	      //Get Index List was successful
	      IF #instOpcUaNamespaceGIL.Done THEN
	        //Check StatusList
	        FOR #tempIndex := 0 TO UDINT_TO_INT(CountOfElements(#namespaceUris) - 1) DO
	          IF #statOpcUaStatusLists.#namespaceGIL[#tempIndex] <> 16#0 THEN
	            #statOpcUaRequests.NGIL := FALSE;
	            // => OUT
	            #statDiagnostics.status := #ERR_NGIL_SL;
	            #statDiagnostics.subfunctionStatus := #statOpcUaStatusLists.namespaceGIL[#tempIndex];
	            // error during NGIL call --> connection establishment failed
	            #statState := #STATE_CONNECT;
	            EXIT;
	          END_IF;
	        END_FOR;
	        #statOpcUaRequests.NGIL := FALSE;
	        IF NOT #statDiagnostics.status.%X15 THEN
	          //Count up statNamespaceGetIndexCount
	          #statDiagCounter.NamespaceReg += 1;
	          //statNamespaceIndexesSet
	          #statRegisteredLists.NamespaceIndexes := TRUE;
	          //=>OUT
	          //Next Step
	          #statState := #STATE_NODE_GET_HANDLE_LIST;
	        ELSE
	          #statCheckConnectionStatus := TRUE;
	        END_IF;
	      END_IF;
	    END_REGION
	    
	  #STATE_NODE_GET_HANDLE_LIST:
	    REGION Handle NodeId lists
	      //Trigger NodeHandleList SFBs
	      IF NOT #statRegisteredLists.Write AND #writeNodeIds <> NULL AND #writeNodeHdls <> NULL THEN
	        #statOpcUaRequests.writeGHL := TRUE;
	        #statDiagnostics.status := #STATUS_BUSY;
	      ELSE
	        IF NOT #statRegisteredLists.Read AND #readNodeIds <> NULL AND #readNodeHdls <> NULL THEN
	          #statOpcUaRequests.readGHL := TRUE;
	          #statDiagnostics.status := #STATUS_BUSY;
	        ELSE
	          IF NOT #statRegisteredLists.Methods AND #methodNodeIds <> NULL AND #methodHdls <> NULL AND #objNodeIds <> NULL THEN
	            #statOpcUaRequests.methodsGHL := TRUE;
	            #statDiagnostics.status := #STATUS_BUSY;
	          ELSE
	            #statState := #STATE_CONNECTED;
	            #statBusy := FALSE;
	            #statDiagnostics.status := #STATUS_IDLE;
	          END_IF;
	        END_IF;
	      END_IF;
	      
	      REGION Handle ReadList
	        //Read Node Get Handle List was not successful
	        IF #InstOpcUaGHLRead.Error THEN
	          //--> Call ConnectionGetStatus if Status = "16#800D0000"
	          IF #InstOpcUaGHLRead.Status = #STATUS_SERVER_NOT_CONNECTED THEN
	            #statCheckConnectionStatus := TRUE;
	          ELSE
	            //#statCase := #STATE_CONNECT;
	            #statState := #STATE_CONNECTED;
	          END_IF;
	          #statOpcUaRequests.readGHL := FALSE;
	          // => OUT
	          #statDiagnostics.status := #ERR_R_GHL;
	          #statDiagnostics.subfunctionStatus := #InstOpcUaGHLRead.Status;
	        END_IF;
	        
	        //Read Node Get Handle List was successful
	        IF #InstOpcUaGHLRead.Done THEN
	          //Check StatusList
	          FOR #tempIndex := 0 TO UDINT_TO_INT(CountOfElements(#readNodeIds) - 1) DO
	            IF #statOpcUaStatusLists.#readGHL[#tempIndex] <> 16#0 THEN
	              // => OUT
	              #statBusy := FALSE;
	              #statDiagnostics.status := #ERR_R_GHL_SL;
	              #statDiagnostics.subfunctionStatus := #statOpcUaStatusLists.#readGHL[#tempIndex];
	              EXIT;
	            END_IF;
	          END_FOR;
	          #statOpcUaRequests.readGHL := FALSE;
	          // Count up statRegisterCount
	          #statDiagCounter.RegisterRead += 1;
	          // Nodes are registered
	          #statRegisteredLists.Read := TRUE;
	        END_IF;
	      END_REGION
	      REGION Handle Write List
	        //Write Node Get Handle List was not successful
	        IF #instOpcUaGHLWrite.Error THEN
	          //--> Call ConnectionGetStatus if Status = "16#800D0000"
	          IF #instOpcUaGHLWrite.Status = #STATUS_SERVER_NOT_CONNECTED THEN
	            #statCheckConnectionStatus := TRUE;
	          ELSE
	            //#statCase := #STATE_CONNECT;
	            #statState := #STATE_CONNECTED;
	          END_IF;
	          #statOpcUaRequests.writeGHL := FALSE;
	          // => OUT
	          #statDiagnostics.status := #ERR_W_GHL;
	          #statDiagnostics.subfunctionStatus := #instOpcUaGHLWrite.Status;
	        END_IF;
	        
	        //Write Node Get Handle List was successful
	        IF #instOpcUaGHLWrite.Done THEN
	          //Check StatusList
	          FOR #tempIndex := 0 TO UDINT_TO_INT(CountOfElements(#writeNodeIds) - 1) DO
	            IF #statOpcUaStatusLists.#writeGHL[#tempIndex] <> 16#0 THEN
	              // => OUT
	              #statBusy := FALSE;
	              #statDiagnostics.status := #ERR_W_GHL_SL;
	              #statDiagnostics.subfunctionStatus := #statOpcUaStatusLists.#writeGHL[#tempIndex];
	              //#statCase := #STATE_CONNECT;
	              EXIT;
	            END_IF;
	          END_FOR;
	          #statOpcUaRequests.writeGHL := FALSE;
	          // Count up statRegisterCount
	          #statDiagCounter.RegisterWrite += 1;
	          // Nodes are registered
	          #statRegisteredLists.Write := TRUE;
	        END_IF;
	      END_REGION
	      
	      REGION Handle MethodList
	        //Method Get HandleList was not successful
	        IF #instOpcUaGHLMethods.Error THEN
	          //--> Call ConnectionGetStatus if Status = "16#800D0000"
	          IF #instOpcUaGHLMethods.Status = #STATUS_SERVER_NOT_CONNECTED THEN
	            #statCheckConnectionStatus := TRUE;
	          ELSE
	            //#statCase := #STATE_CONNECT;
	            #statState := #STATE_CONNECTED;
	          END_IF;
	          #statOpcUaRequests.methodsGHL := FALSE;
	          // => OUT
	          #statDiagnostics.status := #ERR_M_GHL;
	          #statDiagnostics.subfunctionStatus := #instOpcUaGHLMethods.Status;
	        END_IF;
	        
	        //Method Get Handle List was successful
	        IF #instOpcUaGHLMethods.Done THEN
	          //Check StatusList
	          FOR #tempIndex := 0 TO UDINT_TO_INT(CountOfElements(#methodNodeIds) - 1) DO
	            IF #statOpcUaStatusLists.#methodGHL[#tempIndex] <> 16#0 THEN
	              // => OUT
	              #statBusy := FALSE;
	              #statDiagnostics.status := #ERR_M_GHL_SL;
	              #statDiagnostics.subfunctionStatus := #statOpcUaStatusLists.#methodGHL[#tempIndex];
	              EXIT;
	            END_IF;
	          END_FOR;
	          #statOpcUaRequests.methodsGHL := FALSE;
	          // Count up statRegisterCount
	          #statDiagCounter.RegisterMethods += 1;
	          // Nodes are registered
	          #statRegisteredLists.Methods := TRUE;
	        END_IF;
	      END_REGION
	      
	    END_REGION
	    
	  #STATE_CONNECTED:
	    
	    REGION Command and Idle
	      //Idle as long as no Command was triggered
	      IF NOT #statBusy AND NOT #read AND NOT #write AND NOT #callMethod AND NOT #statCheckConnectionStatus THEN
	        #statDone := FALSE;
	        #statDiagnostics.status := #STATUS_IDLE;
	      END_IF;
	      //OPC_UA_GetStatus function is called cyclically, so the connection is monitored
	      #instCycDiag.TON(IN := NOT #statCycDiagTrigger,
	                       PT := #CYC_TIME_GCS);
	      #statCycDiagTrigger := FALSE;
	      IF #instCycDiag.Q AND NOT #statRHLTrigger AND NOT #tempDisconnectTrigger THEN
	        #statCheckConnectionStatus := TRUE;
	        #statCycDiagTrigger := TRUE;
	      END_IF;
	      
	      REGION Read
	        //Trigger if nodes are registered
	        IF #statRegisteredLists.Read AND #statConnected THEN
	          #tempReadTrigger := #read AND NOT #statOldTriggers.read;
	          #statOldTriggers.read := #read;
	        ELSE
	          IF #read AND #statConnected THEN
	            #statDiagnostics.status := #ERR_RL_NOTREG; //Error no ReadList is registerd Request denied
	            #statDiagnostics.subfunctionStatus := #STATUS_NOT_REGISTERED;
	          ELSE
	            IF NOT #statCheckConnectionStatus THEN
	              #statDiagnostics.status := #STATUS_IDLE; //Wait for Connection Get Status
	            END_IF;
	          END_IF;
	        END_IF;
	        
	        IF #tempReadTrigger THEN
	          #statOpcUaRequests.read := TRUE;
	          #statBusy := TRUE;
	          #statDiagnostics.status := #STATUS_BUSY;
	        ELSE
	          #statOpcUaRequests.read := FALSE;
	        END_IF;
	        //Error
	        IF #instOpcUaReadList.Error THEN
	          //--> Call ConnectionGetStatus if Status = "16#800D0000"
	          IF #instOpcUaReadList.Status = #STATUS_SERVER_NOT_CONNECTED THEN
	            #statCheckConnectionStatus := TRUE;
	          END_IF;
	          #statOpcUaRequests.read := FALSE;
	          // => OUT
	          #statBusy := FALSE;
	          #statDiagnostics.status := #ERR_RL;
	          #statDiagnostics.subfunctionStatus := #instOpcUaReadList.Status;
	        END_IF;
	        
	        //Done
	        IF #instOpcUaReadList.Done THEN
	          //Check StatusList
	          FOR #tempIndex := 0 TO UDINT_TO_INT(CountOfElements(#readNodeIds) - 1) DO
	            IF #statOpcUaStatusLists.#readList[#tempIndex] <> 16#0 THEN
	              // => OUT
	              #statDone := FALSE;
	              #statBusy := FALSE;
	              #statDiagnostics.status := #ERR_RL_SL;
	              #statDiagnostics.subfunctionStatus := #statOpcUaStatusLists.readList[#tempIndex];
	              EXIT;
	            END_IF;
	          END_FOR;
	          #statOpcUaRequests.read := FALSE;
	          // => OUT
	          IF NOT #statDiagnostics.status.%X15 THEN
	            #statDone := TRUE;
	            #statBusy := FALSE;
	            #statDiagnostics.status := #STATUS_DONE;
	            //Count up statReadCount
	            #statDiagCounter.Read += 1;
	            //--> Nodes are read continously ...
	          END_IF;
	        END_IF;
	      END_REGION
	      
	      REGION Write
	        //Trigger if nodes are registered
	        IF #statRegisteredLists.Write AND #statConnected THEN
	          #tempWriteTrigger := #write AND NOT #statOldTriggers.write;
	          #statOldTriggers.write := #write;
	        ELSE
	          IF #write AND #statConnected THEN
	            #statDiagnostics.status := #ERR_WL_NOTREG; //Error no WriteList is registerd Request denied
	            #statDiagnostics.subfunctionStatus := #STATUS_NOT_REGISTERED;
	          ELSE
	            IF NOT #statCheckConnectionStatus THEN
	              #statDiagnostics.status := #STATUS_IDLE; //Wait for Connection Get Status
	            END_IF;
	          END_IF;
	        END_IF;
	        
	        IF #tempWriteTrigger THEN
	          #statOpcUaRequests.write := TRUE;
	          #statBusy := TRUE;
	          #statDiagnostics.status := #STATUS_BUSY;
	        ELSE
	          #statOpcUaRequests.write := FALSE;
	        END_IF;
	        //Error
	        IF #instOpcUaWriteList.Error THEN
	          //--> Call ConnectionGetStatus if Status = "16#800D0000"
	          IF #instOpcUaWriteList.Status = #STATUS_SERVER_NOT_CONNECTED THEN
	            #statCheckConnectionStatus := TRUE;
	          END_IF;
	          #statOpcUaRequests.write := FALSE;
	          // => OUT
	          #statBusy := FALSE;
	          #statDiagnostics.status := #ERR_WL;
	          #statDiagnostics.subfunctionStatus := #instOpcUaWriteList.Status;
	        END_IF;
	        
	        //Done
	        IF #instOpcUaWriteList.Done THEN
	          //Check StatusList
	          FOR #tempIndex := 0 TO UDINT_TO_INT(CountOfElements(#writeNodeIds) - 1) DO
	            IF #statOpcUaStatusLists.#writeList[#tempIndex] <> 16#0 THEN
	              // => OUT
	              #statDone := FALSE;
	              #statBusy := FALSE;
	              #statDiagnostics.status := #ERR_WL_SL;
	              #statDiagnostics.subfunctionStatus := #statOpcUaStatusLists.#writeList[#tempIndex];
	              EXIT;
	            END_IF;
	          END_FOR;
	          
	          #statOpcUaRequests.write := FALSE;
	          // => OUT
	          IF NOT #statDiagnostics.status.%X15 THEN
	            #statDone := TRUE;
	            #statBusy := FALSE;
	            #statDiagnostics.status := #STATUS_DONE;
	            //Count up statwriteCount
	            #statDiagCounter.Write += 1;
	            //--> Nodes are write continously ...
	          END_IF;
	        END_IF;
	      END_REGION
	      
	      REGION Method Call
	        //Trigger if methods are registered
	        IF #statRegisteredLists.Methods AND #statConnected THEN
	          #tempMethodCallTrigger := #callMethod AND NOT #statOldTriggers.callMethod;
	          #statOldTriggers.callMethod := #callMethod;
	        ELSE
	          IF #callMethod AND #statConnected THEN
	            #statDiagnostics.status := #ERR_MC_NOTREG; //Error no MethodList is registerd Request denied
	            #statDiagnostics.subfunctionStatus := #STATUS_NOT_REGISTERED;
	          ELSE
	            IF NOT #statCheckConnectionStatus THEN
	              #statDiagnostics.status := #STATUS_IDLE; //Wait for Connection Get Status
	            END_IF;
	          END_IF;
	        END_IF;
	        
	        IF #tempMethodCallTrigger THEN
	          IF #methodHdlIndex <= #MAX_LENGTH_METHOD_INDEX THEN
	            #statMethodHdlId := #methodHdlIndex * 0;
	            //Define statMethodHdl for the input methodHdlIndex choosen index of MethodList
	            #tempRetVal := Serialize(SRC_VARIABLE := #methodHdls,
	                                     DEST_ARRAY => #statSerializeMethodHdls,
	                                     POS := #statMethodHdlId);
	            IF #tempRetVal <> 0 THEN
	              #statDiagnostics.status := #ERR_MC_SERIALIZE;
	              #statDiagnostics.subfunctionStatus := INT_TO_WORD(#tempRetVal);
	            ELSE
	              #statMethodHdlId := #methodHdlIndex * 4;
	              #statMethodHdl.%B0 := #statSerializeMethodHdls[#statMethodHdlId + 3];
	              #statMethodHdl.%B1 := #statSerializeMethodHdls[#statMethodHdlId + 2];
	              #statMethodHdl.%B2 := #statSerializeMethodHdls[#statMethodHdlId + 1];
	              #statMethodHdl.%B3 := #statSerializeMethodHdls[#statMethodHdlId];
	              //Start Method Call
	              #statOpcUaRequests.methodCall := TRUE;
	              #statBusy := TRUE;
	              #statDiagnostics.status := #STATUS_BUSY;
	            END_IF;
	          ELSE
	            //Error handling for Method Handle Index
	            #statDiagnostics.status := #ERR_MC_INDEX_OO_RANGE;
	            #statDiagnostics.subfunctionStatus := INT_TO_WORD(#MAX_LENGTH_METHOD_INDEX);
	          END_IF;
	        ELSE
	          #statOpcUaRequests.methodCall := FALSE;
	        END_IF;
	        //Error
	        IF #instOpcUaMethodCall.Error THEN
	          //--> Call ConnectionGetStatus if Status = "16#800D0000"
	          IF #instOpcUaMethodCall.Status = #STATUS_SERVER_NOT_CONNECTED THEN
	            #statCheckConnectionStatus := TRUE;
	          END_IF;
	          #statOpcUaRequests.methodCall := FALSE;
	          // => OUT
	          #statBusy := FALSE;
	          #statDiagnostics.status := #ERR_MC;
	          #statDiagnostics.subfunctionStatus := #instOpcUaMethodCall.Status;
	        END_IF;
	        
	        //Done
	        IF #instOpcUaMethodCall.Done THEN
	          //Check MethodResult
	          IF #statMethodResult <> 0 THEN
	            #statDone := FALSE;
	            #statBusy := FALSE;
	            #statDiagnostics.status := #ERR_MC_RESULT;
	            #statDiagnostics.subfunctionStatus := #statMethodResult;
	          END_IF;
	          
	          #statOpcUaRequests.methodCall := FALSE;
	          
	          IF NOT #statDiagnostics.status.%X15 THEN
	            // => OUT
	            #statDone := TRUE;
	            #statBusy := FALSE;
	            #statDiagnostics.status := #STATUS_DONE;
	            //Count up statwriteCount
	            #statDiagCounter.MethodCall += 1;
	          END_IF;
	          //--> Methods can be called continously ...
	        END_IF;
	      END_REGION
	      
	      REGION Disconnect Trigger
	        // Trigger to release handles if OPC UA connection should be disconnected
	        #tempClearSessionTrigger := NOT #enable AND #statOldTriggers.clearSession;
	        #statOldTriggers.clearSession := #enable;
	        
	        IF #tempClearSessionTrigger THEN
	          #statBusy := TRUE;
	          #statRHLTrigger := TRUE;
	          #statState := #STATE_DISCONNECT;
	          #statDiagnostics.status := #STATUS_BUSY;
	        END_IF;
	      END_REGION
	    END_REGION
	    
	  #STATE_DISCONNECT:
	    REGION Clear Session
	      //If Disconnect requested, release nodes -> disconnect established connection
	      //-------DISCONNECT HANDLING------------
	      //--------------------------------------
	      
	      IF #statRHLTrigger THEN
	        IF #statRegisteredLists.Write AND #writeNodeIds <> NULL AND #writeNodeHdls <> NULL THEN
	          #statOpcUaRequests.writeRHL := TRUE;
	        ELSE
	          IF #statRegisteredLists.Read AND #readNodeIds <> NULL AND #readNodeHdls <> NULL THEN
	            #statOpcUaRequests.readRHL := TRUE;
	          ELSE
	            IF #statRegisteredLists.Methods AND #methodNodeIds <> NULL AND #methodHdls <> NULL AND #objNodeIds <> NULL THEN
	              #statOpcUaRequests.methodsRHL := TRUE;
	            ELSE
	              #statRHLTrigger := FALSE;
	            END_IF;
	          END_IF;
	        END_IF;
	      END_IF;
	      REGION Release ReadList
	        //Release Handle List of Read Nodes was not successful
	        IF #InstOpcUaRHLRead.Error THEN
	          //--> Call ConnectionGetStatus if Status = "16#800D0000" or "16#80AE0000"
	          IF #InstOpcUaRHLRead.Status = #STATUS_SERVER_NOT_CONNECTED
	            OR #InstOpcUaRHLRead.Status = #STATUS_BAD_CONNECTION_CLOSED
	            
	            OR #InstOpcUaRHLRead.Status = #STATUS_BAD_INVALID_STATE
	            
	          THEN
	            #statCheckConnectionStatus := TRUE;
	            
	            #statRegisteredLists.Read := FALSE;
	            
	          END_IF;
	          #statOpcUaRequests.readRHL := FALSE;
	          // => OUT
	          #statDiagnostics.status := #ERR_R_RHL;
	          #statDiagnostics.subfunctionStatus := #InstOpcUaRHLRead.Status;
	        END_IF;
	        
	        //Release Handle List of Read Nodes was successful
	        IF #InstOpcUaRHLRead.Done THEN
	          //Check StatusList
	          FOR #tempIndex := 0 TO UDINT_TO_INT(CountOfElements(#readNodeIds) - 1) DO
	            IF #statOpcUaStatusLists.#readRHL[#tempIndex] <> 16#0 THEN
	              // => OUT
	              #statDone := FALSE;
	              #statDiagnostics.status := #ERR_R_RHL_SL;
	              #statDiagnostics.subfunctionStatus := #statOpcUaStatusLists.readRHL[#tempIndex];
	              EXIT;
	            END_IF;
	          END_FOR;
	          #statOpcUaRequests.readRHL := FALSE;
	          #statRegisteredLists.Read := FALSE;
	          IF NOT #statDiagnostics.status.%X15 THEN
	            // => OUT
	            #statDiagnostics.status := #STATUS_DONE;
	            //--> Nodes are released
	          END_IF;
	        END_IF;
	      END_REGION
	      
	      REGION Release WriteList
	        //Release Handle List of Write Nodes was not successful
	        IF #instOpcUaRHLWrite.Error THEN
	          //--> Call ConnectionGetStatus if Status = "16#800D0000" or "16#80AE0000"
	          IF #instOpcUaRHLWrite.Status = #STATUS_SERVER_NOT_CONNECTED
	            OR #instOpcUaRHLWrite.Status = #STATUS_BAD_CONNECTION_CLOSED
	            
	            OR #instOpcUaRHLWrite.Status = #STATUS_BAD_INVALID_STATE
	            
	          THEN
	            #statCheckConnectionStatus := TRUE;
	            
	            #statRegisteredLists.Write := FALSE;
	            
	          END_IF;
	          #statOpcUaRequests.writeRHL := FALSE;
	          // => OUT
	          #statDiagnostics.status := #ERR_W_RHL;
	          #statDiagnostics.subfunctionStatus := #instOpcUaRHLWrite.Status;
	        END_IF;
	        
	        //Release Handle List of Write Nodes was successful
	        IF #instOpcUaRHLWrite.Done THEN
	          //Check StatusList
	          FOR #tempIndex := 0 TO UDINT_TO_INT(CountOfElements(#writeNodeIds) - 1) DO
	            IF #statOpcUaStatusLists.writeRHL[#tempIndex] <> 16#0 THEN
	              // => OUT
	              #statDone := FALSE;
	              #statDiagnostics.status := #ERR_W_RHL_SL;
	              #statDiagnostics.subfunctionStatus := #statOpcUaStatusLists.#writeRHL[#tempIndex];
	              EXIT;
	            END_IF;
	          END_FOR;
	          #statOpcUaRequests.writeRHL := FALSE;
	          #statRegisteredLists.Write := FALSE;
	          IF NOT #statDiagnostics.status.%X15 THEN
	            // => OUT
	            #statDiagnostics.status := #STATUS_DONE;
	            //--> Nodes are released
	          END_IF;
	        END_IF;
	      END_REGION
	      
	      REGION Release MethodList
	        //Release Handle List of Methods was not successful
	        IF #instOpcUaRHLMethods.Error THEN
	          //--> Call ConnectionGetStatus if Status = "16#800D0000" or "16#80AE0000"
	          IF #instOpcUaRHLMethods.Status = #STATUS_SERVER_NOT_CONNECTED
	            OR #instOpcUaRHLMethods.Status = #STATUS_BAD_CONNECTION_CLOSED
	            
	            OR #instOpcUaRHLMethods.Status = #STATUS_BAD_INVALID_STATE
	              
	          THEN
	            #statCheckConnectionStatus := TRUE;
	            
	            #statRegisteredLists.Methods := FALSE;
	            
	          END_IF;
	          #statOpcUaRequests.methodsRHL := FALSE;
	          // => OUT
	          #statDiagnostics.status := #ERR_M_RHL;
	          #statDiagnostics.subfunctionStatus := #instOpcUaRHLMethods.Status;
	        END_IF;
	        
	        //Release Handle List of Methods was successful
	        IF #instOpcUaRHLMethods.Done THEN
	          //Check StatusList
	          FOR #tempIndex := 0 TO UDINT_TO_INT(CountOfElements(#methodNodeIds) - 1) DO
	            IF #statOpcUaStatusLists.#methodRHL[#tempIndex] <> 16#0 THEN
	              // => OUT
	              #statDone := FALSE;
	              #statDiagnostics.status := #ERR_M_RHL_SL;
	              #statDiagnostics.subfunctionStatus := #statOpcUaStatusLists.#methodRHL[#tempIndex];
	              EXIT;
	            END_IF;
	          END_FOR;
	          #statOpcUaRequests.methodsRHL := FALSE;
	          #statRegisteredLists.Methods := FALSE;
	          IF NOT #statDiagnostics.status.%X15 THEN
	            // => OUT
	            #statDiagnostics.status := #STATUS_DONE;
	            //--> Nodes are released
	          END_IF;
	        END_IF;
	      END_REGION
	      
	      REGION Disconnect
	        // disconnect trigger, if all nodes and methods are deregistered
	        #tempDisconnectTrigger := NOT #statRegisteredLists.Read AND NOT #statRegisteredLists.Write AND NOT #statRegisteredLists.Methods AND NOT #statOldTriggers.disconnect;
	        #statOldTriggers.disconnect := NOT #statRegisteredLists.Read AND NOT #statRegisteredLists.Write AND NOT #statRegisteredLists.Methods;
	        IF #tempDisconnectTrigger THEN
	          IF #statConnectionHdl <> 16#0 THEN
	            #statOpcUaRequests.disconnect := TRUE;
	            //set FB Outputs
	            #statDiagnostics.status := #STATUS_BUSY;
	          ELSE
	            #statState := #STATE_CONNECT;
	            //Error No connection established
	          END_IF;
	        ELSE
	          #statOpcUaRequests.disconnect := FALSE;
	        END_IF;
	        
	        //Error at connection establishment
	        IF #instOpcUaDisconnect.Error THEN
	          #statBusy := FALSE;
	          #statDiagnostics.status := #ERR_DISCON;
	          #statDiagnostics.subfunctionStatus := #instOpcUaDisconnect.Status;
	          #statCheckConnectionStatus := TRUE;
	        END_IF;
	        
	        //Disconnect was successful
	        IF #instOpcUaDisconnect.Done THEN
	          #statConnected := FALSE;
	          #statDone := FALSE;
	          #statRegisteredLists.NamespaceIndexes := FALSE;
	          #statBusy := FALSE;
	          #statOpcUaRequests.disconnect := FALSE;
	          #statConnectionHdl := 0;
	          
	          IF NOT #statDiagnostics.status.%X15 THEN
	            #statDiagnostics.status := #STATUS_DONE;
	          END_IF;
	          //reset positive edges of functions
	          #statOldTriggers.read := FALSE;
	          #statOldTriggers.write := FALSE;
	          #statOldTriggers.callMethod := FALSE;
	          #statOldTriggers.disconnect := FALSE;
	          #statOldTriggers.clearSession := FALSE;
	          #statState := #STATE_CONNECT;
	        END_IF;
	      END_REGION
	    END_REGION
	    
	  ELSE  // Statement section ELSE
	    ; //Not reachable
	END_CASE;
	REGION Connection Diagnostics
	  IF #statCheckConnectionStatus AND #enable AND (#statConnected OR #statDiagnostics.subfunctionStatus <> #CGS_CONNECTED)
	  THEN
	    #statOpcUaRequests.conGS := TRUE;
	    IF #instOpcUaConnectionGetStatus.Error THEN
	      #statOpcUaRequests.conGS := FALSE;
	      // => OUT
	      #statBusy := FALSE;
	      #statDiagnostics.status := #ERR_CGS;
	      #statDiagnostics.subfunctionStatus := #instOpcUaConnectionGetStatus.Status;
	    END_IF;
	    //Done
	    IF #instOpcUaConnectionGetStatus.Done THEN
	      //ConnectionStatus+ServerState+ServiceLevel are "Good"
	      IF #instOpcUaConnectionGetStatus.ConnectionStatus = #CGS_CONNECTED
	        AND #instOpcUaConnectionGetStatus.ServerState = #CGS_SS_RUNNING
	        AND #instOpcUaConnectionGetStatus.ServiceLevel = #CGS_SL_GOOD
	      THEN
	        REGION Connection OK
	          #statOpcUaRequests.conGS := FALSE;
	          //Session is reactivated and nodes are still registered --> Next Step --> CommandAndIdle
	          IF #statConnected AND #statRegisteredLists.NamespaceIndexes
	            AND (#statRegisteredLists.Read OR #readNodeIds = NULL)
	            AND (#statRegisteredLists.Write OR #writeNodeIds = NULL)
	            AND (#statRegisteredLists.Methods OR #methodNodeIds = NULL)
	          THEN
	            
	            #statBusy := #statBusy AND
	            (
	            #statOpcUaRequests.read OR #instOpcUaReadList.Busy OR
	            #statOpcUaRequests.write OR #instOpcUaWriteList.Busy OR
	            #statOpcUaRequests.methodCall OR #instOpcUaMethodCall.Busy OR
	            #statOpcUaRequests.readRHL OR #InstOpcUaRHLRead.Busy OR
	            #statOpcUaRequests.writeRHL OR #instOpcUaRHLWrite.Busy OR
	            #statOpcUaRequests.methodsRHL OR #instOpcUaRHLMethods.Busy OR
	            #statOpcUaRequests.disconnect OR #instOpcUaDisconnect.Busy
	            );
	            
	            #statCheckConnectionStatus := FALSE;
	            //Session is reactivated and nodes are not registered yet --> Next Step --> NodeGetHandleList
	          ELSIF #statConnected AND #statRegisteredLists.NamespaceIndexes
	            AND (NOT #statRegisteredLists.Read OR NOT #statRegisteredLists.Write OR NOT #statRegisteredLists.Methods)
	          THEN
	            #statState := #STATE_NODE_GET_HANDLE_LIST;
	            #statCheckConnectionStatus := FALSE;
	            //Session is reactivated and namespaceIndexes are not set yet --> Next Step --> NamespaceGetIndexList
	          ELSIF #statConnected AND NOT #statRegisteredLists.NamespaceIndexes
	            AND (NOT #statRegisteredLists.Read OR NOT #statRegisteredLists.Write OR NOT #statRegisteredLists.Methods)
	          THEN
	            #statState := #STATE_NAMESPACE_GET_INDEX_LIST;
	            #statCheckConnectionStatus := FALSE;
	            //Session is reactivated (but connected bit isn't set) and namespaceIndexes are set and nodes are registered
	            //--> Next Step --> CommandAndIdle
	          ELSIF NOT #statConnected AND #statRegisteredLists.NamespaceIndexes
	            AND (#statRegisteredLists.Read OR #readNodeIds = NULL)
	            AND (#statRegisteredLists.Write OR #writeNodeIds = NULL)
	            AND (#statRegisteredLists.Methods OR #methodNodeIds = NULL)
	          THEN
	            //connected has to be set
	            #statConnected := TRUE;
	            #statBusy := FALSE;
	            #statRHLTrigger := FALSE;
	            #statOpcUaRequests.writeRHL := FALSE;
	            #statOpcUaRequests.readRHL := FALSE;
	            #statOpcUaRequests.methodsRHL := FALSE;
	            #statCheckConnectionStatus := FALSE;
	          END_IF;
	        END_REGION
	      ELSE
	        REGION Connection Defect
	          IF #enable THEN
	            //ConnectionStatus is in Status Connection Error -> Connection has to be monitored
	            IF #instOpcUaConnectionGetStatus.ConnectionStatus = #CGS_CONN_ERROR THEN
	              #statOpcUaRequests.conGS := FALSE;
	              
	              #statCheckConnectionStatus := FALSE;
	              
	              // => OUT
	              #statBusy := FALSE;
	              #statConnected := FALSE;
	              #statDiagnostics.status := #ERR_CGS_CSTATE;
	              #statDiagnostics.subfunctionStatus := UDINT_TO_DWORD(#instOpcUaConnectionGetStatus.ConnectionStatus);
	              //Connection status is in Shutdown -> connection handle has to be released with OPC_UA_Disconnect
	            ELSIF #instOpcUaConnectionGetStatus.ConnectionStatus = #CGS_SHUTDOWN THEN
	              #statOpcUaRequests.conGS := FALSE;
	              #statState := #STATE_CONNECT;
	              #statRegisteredLists.Read := FALSE;
	              #statRegisteredLists.Write := FALSE;
	              #statRegisteredLists.Methods := FALSE;
	              #statCheckConnectionStatus := FALSE;
	              // => OUT
	              #statBusy := FALSE;
	              #statConnected := FALSE;
	              #statDiagnostics.status := #ERR_CGS_CSTATE_SHUTDOWN;
	              #statDiagnostics.subfunctionStatus := UDINT_TO_DWORD(#instOpcUaConnectionGetStatus.ConnectionStatus);
	              
	              //ServerState is not "Good"
	            ELSIF #instOpcUaConnectionGetStatus.ServerState <> #CGS_SS_RUNNING THEN
	              #statOpcUaRequests.conGS := FALSE;
	              // => OUT
	              #statBusy := FALSE;
	              #statConnected := FALSE;
	              #statDiagnostics.status := #ERR_CGS_SSTATE;
	              #statDiagnostics.subfunctionStatus := UDINT_TO_DWORD(#instOpcUaConnectionGetStatus.ServerState);
	              //ServiceLevel is not "Good"
	            ELSIF #instOpcUaConnectionGetStatus.ServiceLevel <> #CGS_SL_GOOD THEN
	              #statOpcUaRequests.conGS := FALSE;
	              // => OUT
	              #statBusy := FALSE;
	              #statDiagnostics.status := #ERR_CGS_SLVL;
	              #statDiagnostics.subfunctionStatus := #instOpcUaConnectionGetStatus.ServiceLevel;
	            END_IF;
	          ELSE
	            //enable is not set -> connection was faulty -> back to case CONNECT
	            //new connection can be set up
	            #statCheckConnectionStatus := FALSE;
	            #statOpcUaRequests.conGS := FALSE;
	            #statRHLTrigger := FALSE;
	            #statRegisteredLists.NamespaceIndexes := FALSE;
	            #statRegisteredLists.Read := FALSE;
	            #statRegisteredLists.Write := FALSE;
	            #statRegisteredLists.Methods := FALSE;
	          END_IF;
	        END_REGION
	      END_IF;
	    END_IF;
	  END_IF;
	END_REGION
	
	REGION Call SFBs
	  //CALL SFB OPC_UA_Connect
	  #instOpcUaConnect(REQ := #statOpcUaRequests.connect,
	                    ServerEndpointUrl := #serverEndpointUrl,
	                    SessionConnectInfo := #connectionInfo,
	                    Timeout := #OPC_UA_FUNCTIONS_TIMEOUT,
	                    ConnectionHdl => #tempConnectionHdl);
	  
	  //set connection handle only once after connection setup
	  IF #instOpcUaConnect.Done THEN
	    #statConnectionHdl := #tempConnectionHdl;
	  END_IF;
	  
	  //CALL SFB OPC_UA_NamespaceGetIndexList 
	  #instOpcUaNamespaceGIL(REQ := #statOpcUaRequests.NGIL,
	                         ConnectionHdl := #statConnectionHdl,
	                         NamespaceUrisCount := UDINT_TO_UINT(CountOfElements(#namespaceUris)),
	                         NamespaceUris := #namespaceUris,
	                         Timeout := #OPC_UA_FUNCTIONS_TIMEOUT,
	                         StatusList := #statOpcUaStatusLists.#namespaceGIL,
	                         NamespaceIndexes := #namespaceIndexes);
	  
	  //CALL SFB OPC_UA_NodeGetHandleList_Read
	  #InstOpcUaGHLRead(REQ := #statOpcUaRequests.readGHL,
	                    ConnectionHdl := #statConnectionHdl,
	                    NodeIDCount := UDINT_TO_UINT(CountOfElements(#readNodeIds)),
	                    NodeIDs := #readNodeIds,
	                    Timeout := #OPC_UA_FUNCTIONS_TIMEOUT,
	                    NamespaceIndexCount := UDINT_TO_UINT(CountOfElements(#namespaceIndexes)),
	                    NamespaceIndexes := #namespaceIndexes,
	                    NodeStatusList := #statOpcUaStatusLists.#readGHL,
	                    NodeHdls := #readNodeHdls);
	  
	  //CALL SFB OPC_UA_NodeGetHandleList_Write
	  #instOpcUaGHLWrite(REQ := #statOpcUaRequests.writeGHL,
	                     ConnectionHdl := #statConnectionHdl,
	                     NodeIDCount := UDINT_TO_UINT(CountOfElements(#writeNodeIds)),
	                     NodeIDs := #writeNodeIds,
	                     Timeout := #OPC_UA_FUNCTIONS_TIMEOUT,
	                     NamespaceIndexCount := UDINT_TO_UINT(CountOfElements(#namespaceIndexes)),
	                     NamespaceIndexes := #namespaceIndexes,
	                     NodeStatusList := #statOpcUaStatusLists.#writeGHL,
	                     NodeHdls := #writeNodeHdls);
	  
	  //CALL SFB OPC_UA_MethodGetHandleList
	  #instOpcUaGHLMethods(REQ := #statOpcUaRequests.methodsGHL,
	                       ConnectionHdl := #statConnectionHdl,
	                       NodeIDCount := UDINT_TO_UINT(CountOfElements(#methodNodeIds)),
	                       ObjectNodeIDs := #objNodeIds,
	                       MethodNodeIDs := #methodNodeIds,
	                       Timeout := #OPC_UA_FUNCTIONS_TIMEOUT,
	                       NamespaceIndexCount := UDINT_TO_UINT(CountOfElements(#namespaceIndexes)),
	                       NamespaceIndexes := #namespaceIndexes,
	                       StatusList := #statOpcUaStatusLists.#methodGHL,
	                       MethodHdls := #methodHdls);
	  
	  //CALL SFB OPC_UA_ReadList
	  #instOpcUaReadList(REQ := #statOpcUaRequests.read,
	                     ConnectionHdl := #statConnectionHdl,
	                     NodeHdlCount := UDINT_TO_UINT(CountOfElements(#readNodeHdls)),
	                     NodeHdls := #readNodeHdls,
	                     Timeout := #OPC_UA_FUNCTIONS_TIMEOUT,
	                     NodeStatusList := #statOpcUaStatusLists.#readList,
	                     TimeStamps := #statOpcUaReadTimeStamps,
	                     Variable := #readData);
	  
	  //CALL SFB OPC_UA_WriteList
	  #instOpcUaWriteList(REQ := #statOpcUaRequests.write,
	                      ConnectionHdl := #statConnectionHdl,
	                      NodeHdlCount := UDINT_TO_UINT(CountOfElements(#writeNodeHdls)),
	                      NodeHdls := #writeNodeHdls,
	                      Timeout := #OPC_UA_FUNCTIONS_TIMEOUT,
	                      NodeStatusList := #statOpcUaStatusLists.#writeList,
	                      Variable := #writeData);
	  
	  //CALL SFB OPC_UA_MethodCall
	  #instOpcUaMethodCall(REQ := #statOpcUaRequests.methodCall,
	                       ConnectionHdl := #statConnectionHdl,
	                       MethodHdl := #statMethodHdl,
	                       Timeout := #OPC_UA_FUNCTIONS_TIMEOUT,
	                       MethodResult := #statMethodResult,
	                       InputArguments := #inputArguments,
	                       OutputArguments := #outputArguments);
	  
	  //CALL SFB OPC_UA_NodeReleaseHandleList_Read
	  #InstOpcUaRHLRead(REQ := #statOpcUaRequests.readRHL,
	                    ConnectionHdl := #statConnectionHdl,
	                    NodeHdlCount := UDINT_TO_UINT(CountOfElements(#readNodeHdls)),
	                    NodeHdls := #readNodeHdls,
	                    Timeout := #OPC_UA_FUNCTIONS_TIMEOUT,
	                    NodeStatusList := #statOpcUaStatusLists.#readRHL);
	  
	  //CALL SFB OPC_UA_NodeReleaseHandleList_Write
	  #instOpcUaRHLWrite(REQ := #statOpcUaRequests.writeRHL,
	                     ConnectionHdl := #statConnectionHdl,
	                     NodeHdlCount := UDINT_TO_UINT(CountOfElements(#writeNodeHdls)),
	                     NodeHdls := #writeNodeHdls,
	                     Timeout := #OPC_UA_FUNCTIONS_TIMEOUT,
	                     NodeStatusList := #statOpcUaStatusLists.#writeRHL);
	  
	  //CALL SFB OPC_UA_MethodReleaseHandleList
	  #instOpcUaRHLMethods(REQ := #statOpcUaRequests.methodsRHL,
	                       ConnectionHdl := #statConnectionHdl,
	                       MethodHdlCount := UDINT_TO_UINT(CountOfElements(#methodHdls)),
	                       MethodHdls := #methodHdls,
	                       Timeout := #OPC_UA_FUNCTIONS_TIMEOUT,
	                       StatusList := #statOpcUaStatusLists.#methodRHL);
	  
	  //CALL SFB OPC_UA_Disconnect
	  #instOpcUaDisconnect(REQ := #statOpcUaRequests.disconnect,
	                       ConnectionHdl := #statConnectionHdl,
	                       Timeout := #OPC_UA_FUNCTIONS_TIMEOUT);
	  
	  //CALL SFB OPC_UA_ConnectionGetStatus
	  #instOpcUaConnectionGetStatus(REQ := #statOpcUaRequests.conGS AND
	                                NOT #instOpcUaConnectionGetStatus.REQ AND
	                                NOT #instOpcUaConnectionGetStatus.Busy AND
	                                NOT #instOpcUaConnectionGetStatus.Done AND
	                                NOT #instOpcUaConnectionGetStatus.Error,
	                                ConnectionHdl := #statConnectionHdl,
	                                Timeout := #OPC_UA_FUNCTIONS_TIMEOUT);
	END_REGION
	
	REGION Set FB Outputs
	  #connected := #statConnected;
	  #done := #statDone;
	  #busy := #statBusy;
	  #error := #statDiagnostics.status.%X15;
	  #connectionHdl := #statConnectionHdl;
	  #status := #statDiagnostics.status;
	  IF #statDiagnostics.status.%X15 THEN
	    #diagnostics := #statDiagnostics;
	  END_IF;
	END_REGION
END_FUNCTION_BLOCK

FUNCTION_BLOCK "2. Call_M000_PRODUCTION_DECLARATION"   // FB2002, LAD
{ S7_Optimized_Access := 'TRUE' }
AUTHOR : bartz
VERSION : 0.1
// stored: AutoNumber false, IsIECCheckEnabled false, IsRetainMemResEnabled false, MemoryReserve 100, SetENOAutomatically false, UDAEnableTagReadback false
   VAR_INPUT
      CYCLE_COUNTER : DInt;   // Production counter
      timeUTC { ExternalAccessible := 'False'; ExternalVisible := 'False'; ExternalWritable := 'False'} : DTL;
   END_VAR
   VAR_IN_OUT
      LOCAL_PART_ARRAY : Variant;   // Local part reference
      LOCAL_PART_WSTRING : Variant;
      LOCAL_TOOL : Variant;   // Local tool reference
      TRACA_REF : Variant;   // Traceability reference
      QUANTITY : Variant;
      STATION_NAME : Variant;
   END_VAR
   VAR
      cycleCounter_temp : DInt;
      LOCAL_PART_OK : WString;
      STATION_NAME_OK : WString;
      datestring : WString;
      READ_TIMESTAMP : DTL;
      aux : Struct
         idx : UInt;
         cnt : UInt;
         sizeCnt : Bool;
         LOCAL_PART_STRING : String;
      END_STRUCT;
   END_VAR
   VAR_TEMP
      retVal : Int;
   END_VAR
BEGIN

REGION Network 1 (SCL): PREPARE LOCAL_PART
   REGION PREPARE LOCAL_PART_ARRAY
       //Local part management - variable can be either wstring OR array of char
       IF #LOCAL_PART_WSTRING <> NULL THEN
           VariantGet(SRC := #LOCAL_PART_WSTRING,
                      DST => #LOCAL_PART_OK);
       ELSE
           IF #LOCAL_PART_ARRAY <> NULL THEN
               #aux.sizeCnt := FALSE;
               //If array of char, the array pass through a filter to delete empty positions
               Chars_TO_Strg(Chars := #LOCAL_PART_ARRAY,
                             pChars := 0,
                             Cnt := 0, //Copy all positions of char array
                             Strg => #aux.LOCAL_PART_STRING);

               //Find the last valid char
               #aux.idx := INT_TO_UINT(LEN(#aux.LOCAL_PART_STRING));

               WHILE #aux.sizeCnt = FALSE DO
                   IF #aux.LOCAL_PART_STRING[#aux.idx] <> ' ' THEN
                       //Set the index of last valid char
                       #aux.cnt := #aux.idx;
                       #aux.sizeCnt := TRUE;
                   ELSE
                       #aux.idx := #aux.idx - 1;
                   END_IF;
               END_WHILE;

               //Convert the array of char in string
               Chars_TO_Strg(Chars := #LOCAL_PART_ARRAY,
                             pChars := 0,
                             Cnt := #aux.cnt, //Copy only the right amount of data
                               Strg => #aux.LOCAL_PART_STRING);
               #LOCAL_PART_OK := STRING_TO_WSTRING(#aux.LOCAL_PART_STRING);
           ELSE
               //"MII_Parameters".M000_Status.error := TRUE;
               "MII_Parameters".M000_Status.status := WSTRING#'NO LOCAL PART DEFINED';
           END_IF;
       END_IF;
   END_REGION
END_REGION

REGION Network 2 (SCL): PREPARE CALL METHOD
   IF #cycleCounter_temp <> #CYCLE_COUNTER THEN

       IF #CYCLE_COUNTER > 0 THEN
           //Normal mode
           IF "MII_Parameters".Connection_Status.opcUaConnected THEN

               //Start attempts counter 
               "MII_Parameters".Connection_Status.aux.nAttemptsTotal := 1;

               //Set argument parameters
               "MII_Interface_Data".MII_METHODS.M000_PRODUCTION_DECLARATION.Inputs.CYCLE_COUNTER := DINT_TO_WSTRING(#CYCLE_COUNTER);
               "MII_Interface_Data".MII_METHODS.M000_PRODUCTION_DECLARATION.Inputs.LOCAL_PART := #LOCAL_PART_OK;

               // When there are more than one station at the machine, the _STn is concatenated to the PLC_ID
               IF #STATION_NAME <> NULL THEN
                   VariantGet(SRC := #STATION_NAME,
                              DST => #STATION_NAME_OK);
                   IF #STATION_NAME_OK <> WSTRING#'' THEN
                       "MII_Interface_Data".MII_METHODS.M000_PRODUCTION_DECLARATION.Inputs.PLC_ID := CONCAT_WSTRING(IN1 := "MII_Parameters".Connection.PLC_ID, IN2 := WSTRING#'_', IN3 := #STATION_NAME_OK);
                   ELSE
                       "MII_Interface_Data".MII_METHODS.M000_PRODUCTION_DECLARATION.Inputs.PLC_ID := "MII_Parameters".Connection.PLC_ID;
                   END_IF;
               ELSE
                   "MII_Interface_Data".MII_METHODS.M000_PRODUCTION_DECLARATION.Inputs.PLC_ID := "MII_Parameters".Connection.PLC_ID;
               END_IF;

               IF NOT "MII_Parameters".Connection.OperationMode THEN
                   "MII_Interface_Data".MII_METHODS.M000_PRODUCTION_DECLARATION.Inputs.PLANT := "MII_Parameters".Connection.PlantID;
               ELSE
                   "MII_Interface_Data".MII_METHODS.M000_PRODUCTION_DECLARATION.Inputs.PLANT := CONCAT(IN1 := "MII_Parameters".Connection.PlantID, IN2 := WSTRING#'_TEST');
               END_IF;

               VariantGet(SRC := #LOCAL_TOOL,
                          DST => "MII_Interface_Data".MII_METHODS.M000_PRODUCTION_DECLARATION.Inputs.LOCAL_TOOL);
               VariantGet(SRC := #TRACA_REF,
                          DST => "MII_Interface_Data".MII_METHODS.M000_PRODUCTION_DECLARATION.Inputs.TRACA_REF);
               VariantGet(SRC := #QUANTITY,
                          DST => "MII_Interface_Data".MII_METHODS.M000_PRODUCTION_DECLARATION.Inputs.QUANTITY);

               // New from version 4a
               #datestring := STRING_TO_WSTRING("LGF_DTLtoString_ISO"("date" := #timeUTC, separator := '-'));
               #datestring := REPLACE(IN1 := #datestring, IN2 := WSTRING#'T', L := 1, P := 11);
               // delete after minute
               #datestring := DELETE(IN := #datestring, L := 6, P := 24);
               "MII_Interface_Data".MII_METHODS.M000_PRODUCTION_DECLARATION.Inputs.TIMESTAMP := #datestring;

               //Set index to Production Declaration
               "1. DMC_setConnection_DB".CallBuffer[0] := TRUE;
               "MII_Parameters".M000_Status.status := WSTRING#'IN PROGRESS';

               //Store new cycle counter value
               #cycleCounter_temp := #CYCLE_COUNTER;

               //Downgraded mode - NOT USED           
          (* ELSE
               //Set argument parameters
               "MII_Parameters".M000_Status.Inputs.CYCLE_COUNTER := DINT_TO_WSTRING(#CYCLE_COUNTER);
               "MII_Parameters".M000_Status.Inputs.PLANT := "MII_Parameters".Connection.PlantID;
               "MII_Parameters".M000_Status.Inputs.PLC_ID := "MII_Parameters".Connection.PLC_ID;
               "MII_Parameters".M000_Status.Inputs.LOCAL_PART := #LOCAL_PART_OK;

               VariantGet(SRC := #LOCAL_TOOL,
                          DST => "MII_Parameters".M000_Status.Inputs.LOCAL_TOOL);
               VariantGet(SRC := #TRACA_REF,
                          DST => "MII_Parameters".M000_Status.Inputs.TRACA_REF);
               VariantGet(SRC := #QUANTITY,
                          DST => "MII_Parameters".M000_Status.Inputs.QUANTITY);

               //HMI MUST RESET THE VARIABLE AFTER STORING THE VALUES
               "MII_Parameters".M000_Status.error := TRUE;
               "MII_Parameters".M000_Status.status := Wstring#'DOWNGRADED';
               #retVal := RD_LOC_T("MII_Parameters".M000_Status.timestamp); *)
           END_IF;
       END_IF;
   END_IF;
END_REGION

REGION Network 3 (SCL): TEST MODE
   // Send pre defined data to DMC to test the communication and declaration
   IF "MII_Parameters".Commands.testProdDeclaration THEN

       //Start attempts counter 
       "MII_Parameters".Connection_Status.aux.nAttemptsTotal := 1;

       //Set standard test arguments
       "MII_Interface_Data".MII_METHODS.M000_PRODUCTION_DECLARATION.Inputs.CYCLE_COUNTER := INT_TO_WSTRING("MII_Parameters".Commands.auxTestProdDeclaration);
       "MII_Interface_Data".MII_METHODS.M000_PRODUCTION_DECLARATION.Inputs.PLANT := CONCAT(IN1 := "MII_Parameters".Connection.PlantID, IN2 := WSTRING#'_TEST');
       "MII_Interface_Data".MII_METHODS.M000_PRODUCTION_DECLARATION.Inputs.PLC_ID := "MII_Parameters".Connection.PLC_ID;
       "MII_Interface_Data".MII_METHODS.M000_PRODUCTION_DECLARATION.Inputs.LOCAL_PART := #LOCAL_PART_OK;

       // New from version 4a
       // 
       #datestring := STRING_TO_WSTRING("LGF_DTLtoString_ISO"("date" := #timeUTC, separator := '-'));
       #datestring := REPLACE(IN1 := #datestring, IN2 := WSTRING#'T', L := 1, P := 11);
       // delete after minute
       #datestring := DELETE(IN := #datestring, L := 6, P := 24);
       "MII_Interface_Data".MII_METHODS.M000_PRODUCTION_DECLARATION.Inputs.TIMESTAMP := #datestring;


       "1. DMC_setConnection_DB".CallBuffer[0] := TRUE;
       "MII_Parameters".M000_Status.status := WSTRING#'IN PROGRESS';
   END_IF;
END_REGION
END_FUNCTION_BLOCK

FUNCTION_BLOCK "6. Call_M004_NTRS"   // FB2006, LAD
{ S7_Optimized_Access := 'TRUE' }
AUTHOR : bartz
VERSION : 0.1
// stored: AutoNumber false, IsIECCheckEnabled false, IsRetainMemResEnabled false, MemoryReserve 100, SetENOAutomatically false, UDAEnableTagReadback false
   VAR_INPUT
      nTRSTag : Bool;
      TIMESTAMP_IN { ExternalAccessible := 'False'; ExternalVisible := 'False'; ExternalWritable := 'False'} : WString;
   END_VAR
   VAR
      nTRSTagTemp : Bool;
   END_VAR
BEGIN

REGION Network 1 (SCL)
   IF #nTRSTag <> #nTRSTagTemp THEN

       "MII_Interface_Data".MII_METHODS.M004_NTRS.Inputs.PLC_ID := "MII_Parameters".Connection.PLC_ID;
       "MII_Interface_Data".MII_METHODS.M004_NTRS.Inputs.PLANT := "MII_Parameters".Connection.PlantID;
       "MII_Interface_Data".MII_METHODS.M004_NTRS.Inputs.STOPPAGE := #nTRSTag;

       // New from version 4a
       "MII_Interface_Data".MII_METHODS.M004_NTRS.Inputs.TIMESTAMP := #TIMESTAMP_IN;

       //Call the method 
       "1. DMC_setConnection_DB".CallBuffer[6] := TRUE;

       #nTRSTagTemp := #nTRSTag;
   END_IF;
END_REGION
END_FUNCTION_BLOCK

FUNCTION_BLOCK "7. Call_M103_PY"   // FB2007, LAD
{ S7_Optimized_Access := 'TRUE' }
AUTHOR : bartz
VERSION : 0.1
// stored: AutoNumber false, IsIECCheckEnabled false, IsRetainMemResEnabled false, MemoryReserve 100, SetENOAutomatically false, UDAEnableTagReadback false
   VAR_INPUT
      PY_ON : Bool;
      PY_DOWN : Bool;
      PY_OFF : Bool;
   END_VAR
   VAR
      PYOnTemp : Bool;
      PYDownTemp : Bool;
      PYOffTemp : Bool;
   END_VAR
BEGIN

REGION Network 1 (SCL)
   IF (#PY_ON <> #PYOnTemp OR #PY_DOWN <> #PYDownTemp OR #PY_OFF <> #PYOffTemp) AND (#PY_ON OR #PY_DOWN OR #PY_OFF) THEN

       "MII_Interface_Data".MII_METHODS.M103_PY.Inputs.PLC_ID := "MII_Parameters".Connection.PLC_ID;
       "MII_Interface_Data".MII_METHODS.M103_PY.Inputs.PLANT := "MII_Parameters".Connection.PlantID;

       "MII_Interface_Data".MII_METHODS.M103_PY.Inputs.PY_ON := #PY_ON;
       "MII_Interface_Data".MII_METHODS.M103_PY.Inputs.PY_DOWN := #PY_DOWN;
       "MII_Interface_Data".MII_METHODS.M103_PY.Inputs.PY_OFF := #PY_OFF;

       //Call the method 
       "1. DMC_setConnection_DB".CallBuffer[7] := TRUE;

       #PYOnTemp := #PY_ON;
       #PYDownTemp := #PY_DOWN;
       #PYOffTemp := #PY_OFF;
   END_IF;
END_REGION
END_FUNCTION_BLOCK

FUNCTION "Concatenate_STRING" : Void   // FC2010, LAD
{ S7_Optimized_Access := 'TRUE' }
VERSION : 0.1
// stored: AutoNumber false, IsIECCheckEnabled false, SetENOAutomatically false, UDAEnableTagReadback false
   VAR_INPUT
      DMC_SAP_REF : Array[1..10] of String[25];
   END_VAR
   VAR_OUTPUT
      String_empty : Bool;
   END_VAR
   VAR_IN_OUT
      DMC_SAP_REf_WSTRING : WString;
   END_VAR
   VAR_TEMP
      concatenate : String;
      Convert : WString;
   END_VAR
   VAR CONSTANT
      Template_string_empty : String := ';;;;;;;;;';
   END_VAR
BEGIN

REGION Network 1 (SCL): Concatenate function
       #concatenate := CONCAT(IN1 := #DMC_SAP_REF[1], IN2 := ';');
       #concatenate := CONCAT(IN1 := #concatenate, IN2 := #DMC_SAP_REF[2]);
       #concatenate := CONCAT(IN1 := #concatenate, IN2 := ';');
       #concatenate := CONCAT(IN1 := #concatenate, IN2 := #DMC_SAP_REF[3]);
       #concatenate := CONCAT(IN1 := #concatenate, IN2 := ';');
       #concatenate := CONCAT(IN1 := #concatenate, IN2 := #DMC_SAP_REF[4]);
       #concatenate := CONCAT(IN1 := #concatenate, IN2 := ';');
       #concatenate := CONCAT(IN1 := #concatenate, IN2 := #DMC_SAP_REF[5]);
       #concatenate := CONCAT(IN1 := #concatenate, IN2 := ';');
       #concatenate := CONCAT(IN1 := #concatenate, IN2 := #DMC_SAP_REF[6]);
       #concatenate := CONCAT(IN1 := #concatenate, IN2 := ';');
       #concatenate := CONCAT(IN1 := #concatenate, IN2 := #DMC_SAP_REF[7]);
       #concatenate := CONCAT(IN1 := #concatenate, IN2 := ';');
       #concatenate := CONCAT(IN1 := #concatenate, IN2 := #DMC_SAP_REF[8]);
       #concatenate := CONCAT(IN1 := #concatenate, IN2 := ';');
       #concatenate := CONCAT(IN1 := #concatenate, IN2 := #DMC_SAP_REF[9]);
       #concatenate := CONCAT(IN1 := #concatenate, IN2 := ';');
       #concatenate := CONCAT(IN1 := #concatenate, IN2 := #DMC_SAP_REF[10]);
END_REGION

REGION Network 2
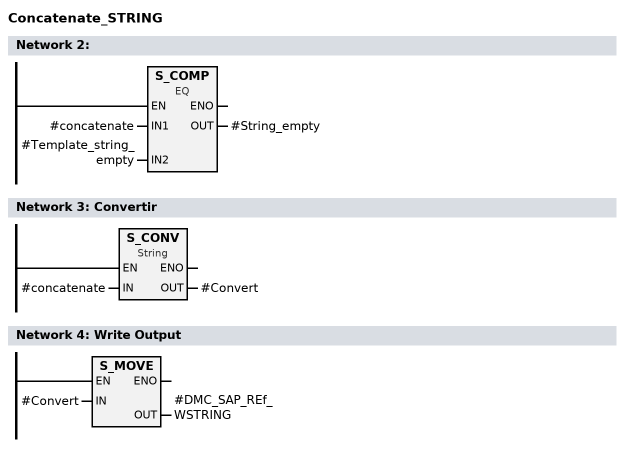
   RUNG wire#powerrail
      { S7_Templates := "[relation := EQ, src_type := String]" } S_COMP(IN1 := #concatenate, IN2 := #Template_string_empty, OUT => #String_empty)
   END_RUNG
   // the same network as SCL:
   S_COMP(IN1 := #concatenate, IN2 := #Template_string_empty, OUT => #String_empty);
END_REGION

REGION Network 3: Convertir
   RUNG wire#powerrail
      { S7_Templates := "[src_type := String, dest_type := WString]" } S_CONV(IN := #concatenate, OUT => #Convert)
   END_RUNG
   // the same network as SCL:
   S_CONV(IN := #concatenate, OUT => #Convert);
END_REGION

REGION Network 4: Write Output
   RUNG wire#powerrail
      S_Move(in := #Convert, out => #DMC_SAP_REf_WSTRING)
   END_RUNG
   // the same network as SCL:
   #DMC_SAP_REf_WSTRING := #Convert;
END_REGION
END_FUNCTION

FUNCTION "Extract_data_DMC" : Void   // FC2011, LAD
{ S7_Optimized_Access := 'TRUE' }
VERSION : 0.1
// stored: AutoNumber false, IsIECCheckEnabled false, SetENOAutomatically false, UDAEnableTagReadback false
   VAR_INPUT
      round : Byte;
      Data_DMC : Array[1.."MaxRoundNumber", 1..10] of "DATA_DMC";
   END_VAR
   VAR_OUTPUT
      DATA_DMC_Extract : Array[1..10] of String[25];
   END_VAR
   VAR_TEMP
      idx : SInt;
      round_idx : SInt;
   END_VAR
BEGIN

REGION Network 1
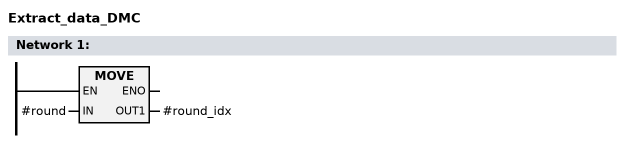
   RUNG wire#powerrail
      Move(in := #round, out1 => #round_idx)
   END_RUNG
   // the same network as SCL:
   #round_idx := #round;
END_REGION

REGION Network 2 (SCL)
   FOR #idx := 1 TO 10 DO
       #DATA_DMC_Extract[#idx] := #Data_DMC[#round_idx, #idx].SAP_REF_PRODUCTION;

   END_FOR;
END_REGION
END_FUNCTION

FUNCTION "FC_DMC" : Void   // FC2012, LAD
{ S7_Optimized_Access := 'TRUE' }
VERSION : 0.1
// stored: AutoNumber false, IsIECCheckEnabled false, SetENOAutomatically false, UDAEnableTagReadback false
   VAR_TEMP
      stationName1 : WString;
      stationName2 : WString;
      Data_DMC : Array[1.."MaxRoundNumber", 1..10] of "DATA_DMC";
      timeUTC : DTL;
      _ret_val : Int;
   END_VAR
BEGIN

REGION Network 1
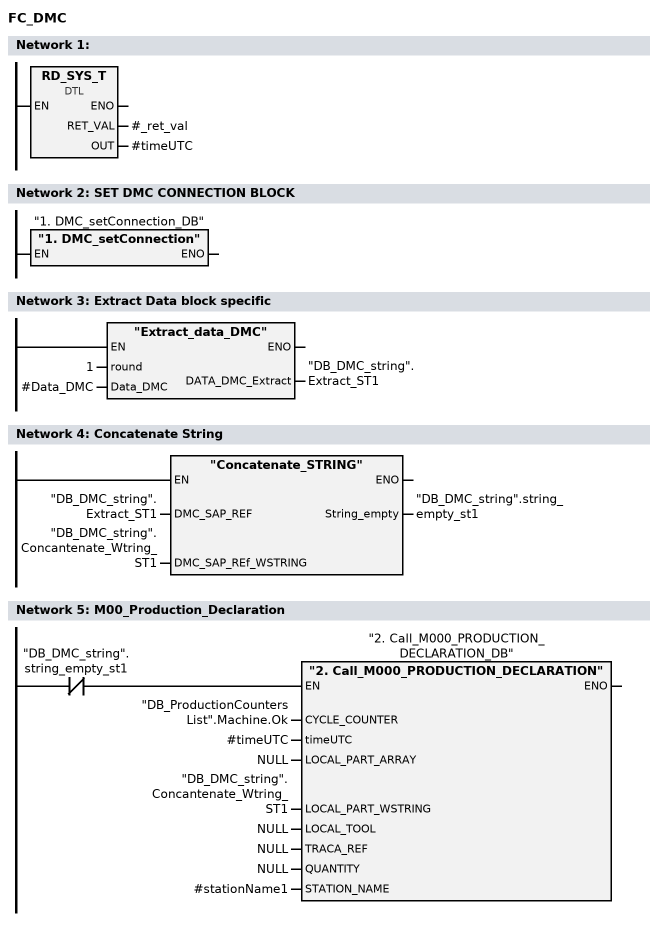
   RUNG wire#powerrail
      { S7_Templates := "date_type := DTL" } RD_SYS_T(RET_VAL => #_ret_val, OUT => #timeUTC)
   END_RUNG
   // the same network as SCL:
   #_ret_val := RD_SYS_T(OUT => #timeUTC);
END_REGION

REGION Network 2: SET DMC CONNECTION BLOCK
   RUNG wire#powerrail
      "1. DMC_setConnection_DB"()
   END_RUNG
   // the same network as SCL:
   "1. DMC_setConnection_DB"();   // "1. DMC_setConnection"
END_REGION

REGION Network 3: Extract Data block specific
   RUNG wire#powerrail
      "Extract_data_DMC"(round := 1, Data_DMC := #Data_DMC, DATA_DMC_Extract => "DB_DMC_string".Extract_ST1)
   END_RUNG
   // the same network as SCL:
   "Extract_data_DMC"(round := 1, Data_DMC := #Data_DMC, DATA_DMC_Extract => "DB_DMC_string".Extract_ST1);
END_REGION

REGION Network 4: Concatenate String
   RUNG wire#powerrail
      "Concatenate_STRING"(DMC_SAP_REF := "DB_DMC_string".Extract_ST1, DMC_SAP_REf_WSTRING := "DB_DMC_string".Concantenate_Wtring_ST1, String_empty => "DB_DMC_string".string_empty_st1)
   END_RUNG
   // the same network as SCL:
   "Concatenate_STRING"(DMC_SAP_REF := "DB_DMC_string".Extract_ST1,
                        DMC_SAP_REf_WSTRING := "DB_DMC_string".Concantenate_Wtring_ST1,
                        String_empty => "DB_DMC_string".string_empty_st1);
END_REGION

REGION Network 5: M00_Production_Declaration
   RUNG wire#powerrail
      I_Contact( "DB_DMC_string".string_empty_st1 )
      "2. Call_M000_PRODUCTION_DECLARATION_DB"(CYCLE_COUNTER := "DB_ProductionCountersList".Machine.Ok, timeUTC := #timeUTC, LOCAL_PART_ARRAY := NULL, LOCAL_PART_WSTRING := "DB_DMC_string".Concantenate_Wtring_ST1, LOCAL_TOOL := NULL, TRACA_REF := NULL, QUANTITY := NULL, STATION_NAME := #stationName1)
   END_RUNG
   // the same network as SCL:
   IF NOT "DB_DMC_string".string_empty_st1 THEN
       "2. Call_M000_PRODUCTION_DECLARATION_DB"(CYCLE_COUNTER := "DB_ProductionCountersList".Machine.Ok,   // "2. Call_M000_PRODUCTION_DECLARATION"
                               timeUTC := #timeUTC,
                               LOCAL_PART_ARRAY := NULL,
                               LOCAL_PART_WSTRING := "DB_DMC_string".Concantenate_Wtring_ST1,
                               LOCAL_TOOL := NULL,
                               TRACA_REF := NULL,
                               QUANTITY := NULL,
                               STATION_NAME := #stationName1);
   END_IF;
END_REGION
END_FUNCTION

FUNCTION_BLOCK "Main_Safety_RTG1"   // FB0, F_LAD
{ S7_Optimized_Access := 'TRUE' }
VERSION : 0.1
// stored: AutoNumber false, IsIECCheckEnabled false, UDAEnableTagReadback false
   VAR
      ACK_GL_Instance : ACK_GL;
      "ESTOP1_3L+" : ESTOP1;
      "FDBACK_A2.7" : FDBACK;
      "ESTOP1_4L+" : ESTOP1;
      "FDBACK_A2.8" : FDBACK;
      "FDBACK_A2.9" : FDBACK;
      "ESTOP1_5L+" : ESTOP1;
      "F_IEC_Timer_3L+" : TON;
      "F_IEC_Timer_4L+" : TON;
      FDBACK_KF101x : FDBACK;
      FDBACK_KM20_KM21 : FDBACK;
   END_VAR
BEGIN

REGION Network 1: ACK_GL
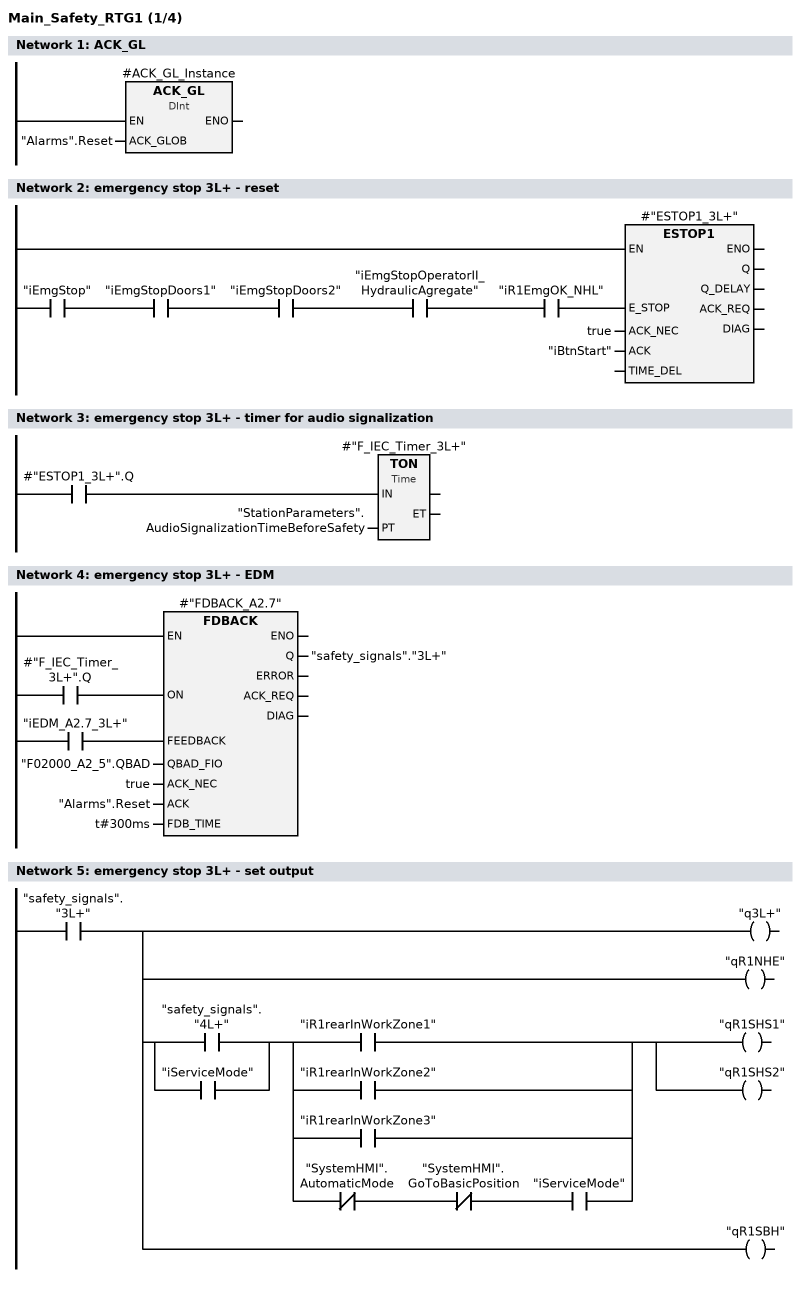
   RUNG wire#powerrail
      { S7_Templates := "codedbool_type := DInt" } #ACK_GL_Instance.ACK_GL(ACK_GLOB := "Alarms".Reset)
   END_RUNG
   // the same network as SCL:
   #ACK_GL_Instance(ACK_GLOB := "Alarms".Reset);   // ACK_GL
END_REGION

REGION Network 2: emergency stop 3L+ - reset
   RUNG wire#powerrail
      #"ESTOP1_3L+".ESTOP1(E_STOP := wire#w1, ACK_NEC := true, ACK := "iBtnStart", TIME_DEL :=, Q =>, Q_DELAY =>, ACK_REQ =>, DIAG =>)
   END_RUNG
   RUNG wire#powerrail
      Contact( "iEmgStop" )
      Contact( "iEmgStopDoors1" )
      Contact( "iEmgStopDoors2" )
      Contact( "iEmgStopOperatorII_HydraulicAgregate" )
      Contact( "iR1EmgOK_NHL" )
   END_RUNG wire#w1
   // the same network as SCL:
   #"ESTOP1_3L+"(E_STOP := "iEmgStop" AND "iEmgStopDoors1" AND "iEmgStopDoors2" AND "iEmgStopOperatorII_HydraulicAgregate" AND "iR1EmgOK_NHL",   // ESTOP1
                 ACK_NEC := true,
                 ACK := "iBtnStart");
END_REGION

REGION Network 3: emergency stop 3L+ - timer for audio signalization
   RUNG wire#powerrail
      Contact( #"ESTOP1_3L+".Q )
      { S7_Templates := "[time_type := Time, codedbool_type := DInt]" } #"F_IEC_Timer_3L+".TON(pt := "StationParameters".AudioSignalizationTimeBeforeSafety, et =>)
   END_RUNG
   // the same network as SCL:
   #"F_IEC_Timer_3L+".TON(IN := #"ESTOP1_3L+".Q, PT := "StationParameters".AudioSignalizationTimeBeforeSafety);
END_REGION

REGION Network 4: emergency stop 3L+ - EDM
   RUNG wire#powerrail
      #"FDBACK_A2.7".FDBACK(ON := wire#w1, FEEDBACK := wire#w2, QBAD_FIO := "F02000_A2_5".QBAD, ACK_NEC := true, ACK := "Alarms".Reset, FDB_TIME := t#300ms, Q => "safety_signals"."3L+", ERROR =>, ACK_REQ =>, DIAG =>)
   END_RUNG
   RUNG wire#powerrail
      Contact( #"F_IEC_Timer_3L+".Q )
   END_RUNG wire#w1
   RUNG wire#powerrail
      Contact( "iEDM_A2.7_3L+" )
   END_RUNG wire#w2
   // the same network as SCL:
   #"FDBACK_A2.7"(ON := #"F_IEC_Timer_3L+".Q,   // FDBACK
                  FEEDBACK := "iEDM_A2.7_3L+",
                  QBAD_FIO := "F02000_A2_5".QBAD,
                  ACK_NEC := true,
                  ACK := "Alarms".Reset,
                  FDB_TIME := t#300ms,
                  Q => "safety_signals"."3L+");
END_REGION

REGION Network 5: emergency stop 3L+ - set output
   RUNG wire#powerrail
      Contact( "safety_signals"."3L+" )
      wire#w1
      Coil( "q3L+" )
   END_RUNG
   RUNG wire#w1
      Coil( "qR1NHE" )
   END_RUNG
   RUNG wire#w1
      Contact( "safety_signals"."4L+" )
      wire#w2
      Contact( "iR1rearInWorkZone1" )
      wire#w3
      Coil( "qR1SHS1" )
   END_RUNG
   RUNG wire#w1
      Contact( "iServiceMode" )
   END_RUNG wire#w2
   RUNG wire#w2
      Contact( "iR1rearInWorkZone2" )
   END_RUNG wire#w3
   RUNG wire#w2
      Contact( "iR1rearInWorkZone3" )
   END_RUNG wire#w3
   RUNG wire#w2
      I_Contact( "SystemHMI".AutomaticMode )
      I_Contact( "SystemHMI".GoToBasicPosition )
      Contact( "iServiceMode" )
   END_RUNG wire#w3
   RUNG wire#w3
      Coil( "qR1SHS2" )
   END_RUNG
   RUNG wire#w1
      Coil( "qR1SBH" )
   END_RUNG
   // the same network as SCL:
   "q3L+" := "safety_signals"."3L+";
   "qR1NHE" := "safety_signals"."3L+";
   "qR1SHS1" := "safety_signals"."3L+" AND ("safety_signals"."4L+" OR "iServiceMode") AND ("iR1rearInWorkZone1" OR "iR1rearInWorkZone2" OR "iR1rearInWorkZone3" OR (NOT "SystemHMI".AutomaticMode AND NOT "SystemHMI".GoToBasicPosition AND "iServiceMode"));
   "qR1SHS2" := "qR1SHS1";
   "qR1SBH" := "safety_signals"."3L+";
END_REGION

REGION Network 6: emergency stop / service doors 4L+ - reset
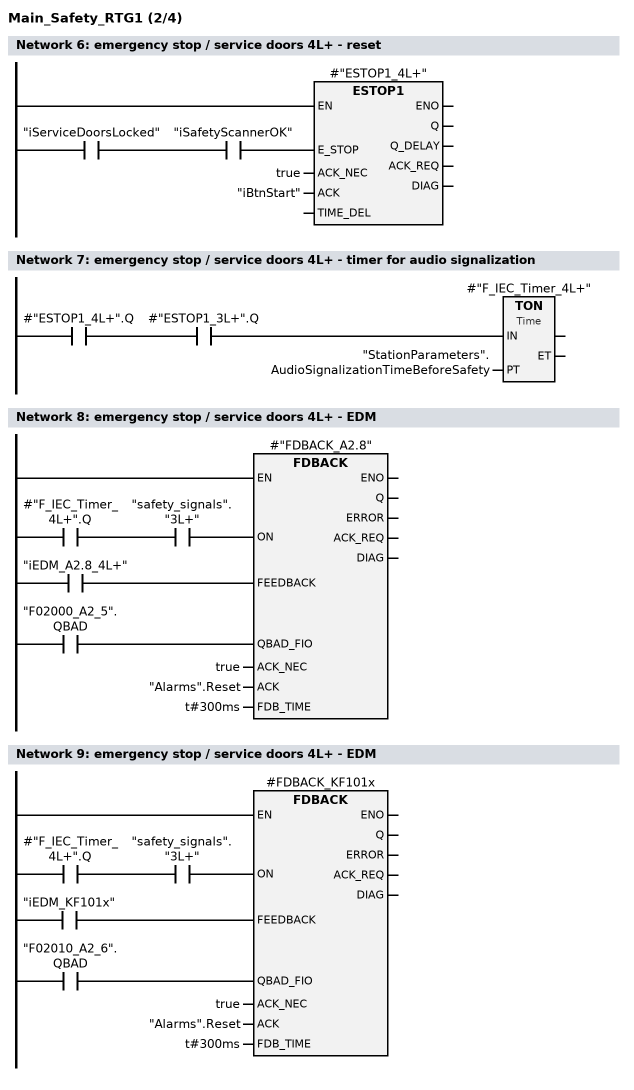
   RUNG wire#powerrail
      #"ESTOP1_4L+".ESTOP1(E_STOP := wire#w1, ACK_NEC := true, ACK := "iBtnStart", TIME_DEL :=, Q =>, Q_DELAY =>, ACK_REQ =>, DIAG =>)
   END_RUNG
   RUNG wire#powerrail
      Contact( "iServiceDoorsLocked" )
      Contact( "iSafetyScannerOK" )
   END_RUNG wire#w1
   // the same network as SCL:
   #"ESTOP1_4L+"(E_STOP := "iServiceDoorsLocked" AND "iSafetyScannerOK", ACK_NEC := true, ACK := "iBtnStart");   // ESTOP1
END_REGION

REGION Network 7: emergency stop / service doors 4L+ - timer for audio signalization
   RUNG wire#powerrail
      Contact( #"ESTOP1_4L+".Q )
      Contact( #"ESTOP1_3L+".Q )
      { S7_Templates := "[time_type := Time, codedbool_type := DInt]" } #"F_IEC_Timer_4L+".TON(pt := "StationParameters".AudioSignalizationTimeBeforeSafety, et =>)
   END_RUNG
   // the same network as SCL:
   #"F_IEC_Timer_4L+".TON(IN := #"ESTOP1_4L+".Q AND #"ESTOP1_3L+".Q,
                          PT := "StationParameters".AudioSignalizationTimeBeforeSafety);
END_REGION

REGION Network 8: emergency stop / service doors 4L+ - EDM
   RUNG wire#powerrail
      #"FDBACK_A2.8".FDBACK(ON := wire#w1, FEEDBACK := wire#w2, QBAD_FIO := wire#w3, ACK_NEC := true, ACK := "Alarms".Reset, FDB_TIME := t#300ms, Q =>, ERROR =>, ACK_REQ =>, DIAG =>)
   END_RUNG
   RUNG wire#powerrail
      Contact( #"F_IEC_Timer_4L+".Q )
      Contact( "safety_signals"."3L+" )
   END_RUNG wire#w1
   RUNG wire#powerrail
      Contact( "iEDM_A2.8_4L+" )
   END_RUNG wire#w2
   RUNG wire#powerrail
      Contact( "F02000_A2_5".QBAD )
   END_RUNG wire#w3
   // the same network as SCL:
   #"FDBACK_A2.8"(ON := #"F_IEC_Timer_4L+".Q AND "safety_signals"."3L+",   // FDBACK
                  FEEDBACK := "iEDM_A2.8_4L+",
                  QBAD_FIO := "F02000_A2_5".QBAD,
                  ACK_NEC := true,
                  ACK := "Alarms".Reset,
                  FDB_TIME := t#300ms);
END_REGION

REGION Network 9: emergency stop / service doors 4L+ - EDM
   RUNG wire#powerrail
      #FDBACK_KF101x.FDBACK(ON := wire#w1, FEEDBACK := wire#w2, QBAD_FIO := wire#w3, ACK_NEC := true, ACK := "Alarms".Reset, FDB_TIME := t#300ms, Q =>, ERROR =>, ACK_REQ =>, DIAG =>)
   END_RUNG
   RUNG wire#powerrail
      Contact( #"F_IEC_Timer_4L+".Q )
      Contact( "safety_signals"."3L+" )
   END_RUNG wire#w1
   RUNG wire#powerrail
      Contact( "iEDM_KF101x" )
   END_RUNG wire#w2
   RUNG wire#powerrail
      Contact( "F02010_A2_6".QBAD )
   END_RUNG wire#w3
   // the same network as SCL:
   #FDBACK_KF101x(ON := #"F_IEC_Timer_4L+".Q AND "safety_signals"."3L+",   // FDBACK
                  FEEDBACK := "iEDM_KF101x",
                  QBAD_FIO := "F02010_A2_6".QBAD,
                  ACK_NEC := true,
                  ACK := "Alarms".Reset,
                  FDB_TIME := t#300ms);
END_REGION

REGION Network 10: emergency stop / service doors 4L+ - set output
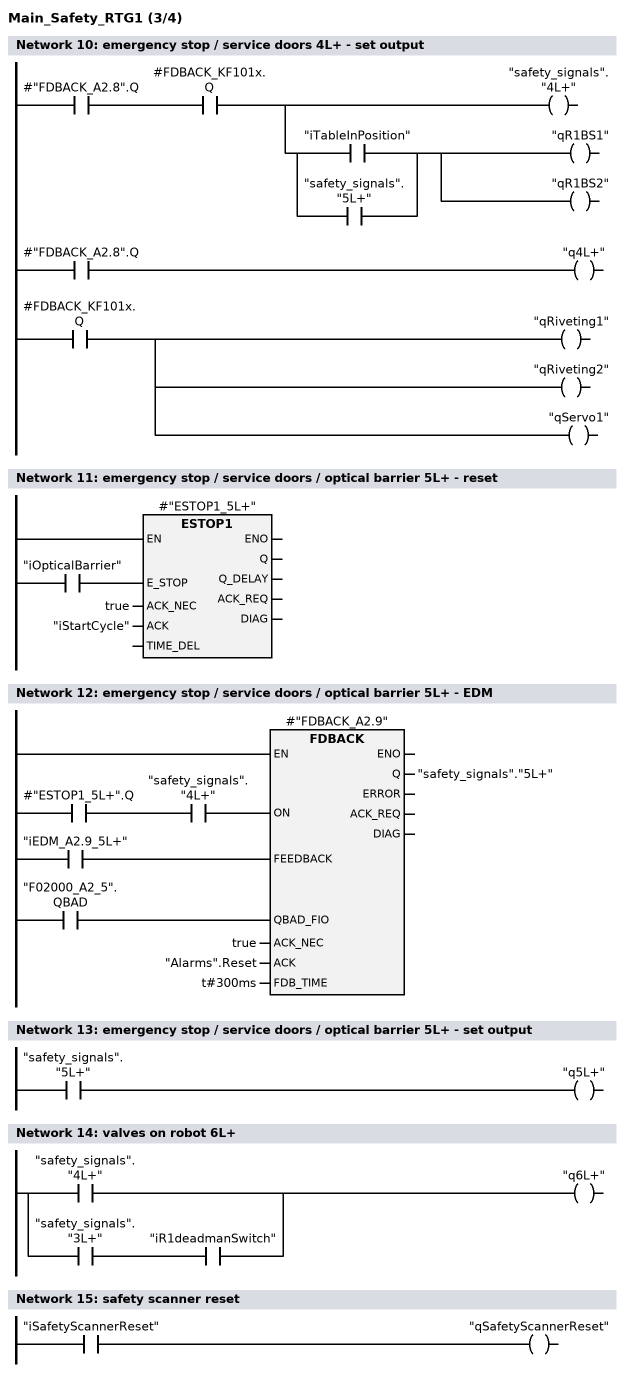
   RUNG wire#powerrail
      Contact( #"FDBACK_A2.8".Q )
      Contact( #FDBACK_KF101x.Q )
      wire#w1
      Coil( "safety_signals"."4L+" )
   END_RUNG
   RUNG wire#w1
      Contact( "iTableInPosition" )
      wire#w2
      Coil( "qR1BS1" )
   END_RUNG
   RUNG wire#w1
      Contact( "safety_signals"."5L+" )
   END_RUNG wire#w2
   RUNG wire#w2
      Coil( "qR1BS2" )
   END_RUNG
   RUNG wire#powerrail
      Contact( #"FDBACK_A2.8".Q )
      Coil( "q4L+" )
   END_RUNG
   RUNG wire#powerrail
      Contact( #FDBACK_KF101x.Q )
      wire#w3
      Coil( "qRiveting1" )
   END_RUNG
   RUNG wire#w3
      Coil( "qRiveting2" )
   END_RUNG
   RUNG wire#w3
      Coil( "qServo1" )
   END_RUNG
   // the same network as SCL:
   "safety_signals"."4L+" := #"FDBACK_A2.8".Q AND #FDBACK_KF101x.Q;
   "qR1BS1" := "safety_signals"."4L+" AND ("iTableInPosition" OR "safety_signals"."5L+");
   "qR1BS2" := "qR1BS1";
   "q4L+" := #"FDBACK_A2.8".Q;
   "qRiveting1" := #FDBACK_KF101x.Q;
   "qRiveting2" := #FDBACK_KF101x.Q;
   "qServo1" := #FDBACK_KF101x.Q;
END_REGION

REGION Network 11: emergency stop / service doors / optical barrier 5L+ - reset
   RUNG wire#powerrail
      #"ESTOP1_5L+".ESTOP1(E_STOP := wire#w1, ACK_NEC := true, ACK := "iStartCycle", TIME_DEL :=, Q =>, Q_DELAY =>, ACK_REQ =>, DIAG =>)
   END_RUNG
   RUNG wire#powerrail
      Contact( "iOpticalBarrier" )
   END_RUNG wire#w1
   // the same network as SCL:
   #"ESTOP1_5L+"(E_STOP := "iOpticalBarrier", ACK_NEC := true, ACK := "iStartCycle");   // ESTOP1
END_REGION

REGION Network 12: emergency stop / service doors / optical barrier 5L+ - EDM
   RUNG wire#powerrail
      #"FDBACK_A2.9".FDBACK(ON := wire#w1, FEEDBACK := wire#w2, QBAD_FIO := wire#w3, ACK_NEC := true, ACK := "Alarms".Reset, FDB_TIME := t#300ms, Q => "safety_signals"."5L+", ERROR =>, ACK_REQ =>, DIAG =>)
   END_RUNG
   RUNG wire#powerrail
      Contact( #"ESTOP1_5L+".Q )
      Contact( "safety_signals"."4L+" )
   END_RUNG wire#w1
   RUNG wire#powerrail
      Contact( "iEDM_A2.9_5L+" )
   END_RUNG wire#w2
   RUNG wire#powerrail
      Contact( "F02000_A2_5".QBAD )
   END_RUNG wire#w3
   // the same network as SCL:
   #"FDBACK_A2.9"(ON := #"ESTOP1_5L+".Q AND "safety_signals"."4L+",   // FDBACK
                  FEEDBACK := "iEDM_A2.9_5L+",
                  QBAD_FIO := "F02000_A2_5".QBAD,
                  ACK_NEC := true,
                  ACK := "Alarms".Reset,
                  FDB_TIME := t#300ms,
                  Q => "safety_signals"."5L+");
END_REGION

REGION Network 13: emergency stop / service doors / optical barrier 5L+ - set output
   RUNG wire#powerrail
      Contact( "safety_signals"."5L+" )
      Coil( "q5L+" )
   END_RUNG
   // the same network as SCL:
   "q5L+" := "safety_signals"."5L+";
END_REGION

REGION Network 14: valves on robot 6L+
   RUNG wire#powerrail
      Contact( "safety_signals"."4L+" )
      wire#w1
      Coil( "q6L+" )
   END_RUNG
   RUNG wire#powerrail
      Contact( "safety_signals"."3L+" )
      Contact( "iR1deadmanSwitch" )
   END_RUNG wire#w1
   // the same network as SCL:
   "q6L+" := "safety_signals"."4L+" OR ("safety_signals"."3L+" AND "iR1deadmanSwitch");
END_REGION

REGION Network 15: safety scanner reset
   RUNG wire#powerrail
      Contact( "iSafetyScannerReset" )
      Coil( "qSafetyScannerReset" )
   END_RUNG
   // the same network as SCL:
   "qSafetyScannerReset" := "iSafetyScannerReset";
END_REGION

REGION Network 16: tool selection for robot - mandatory, but not used
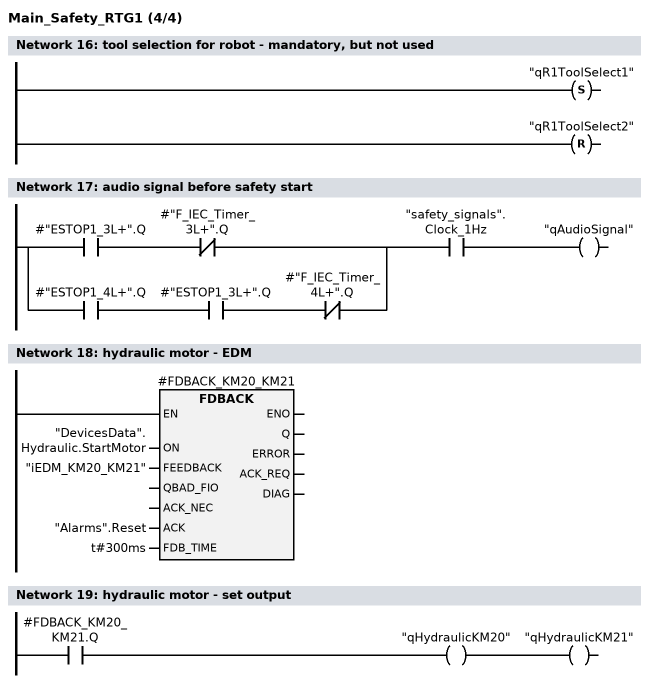
   RUNG wire#powerrail
      S_Coil( "qR1ToolSelect1" )
   END_RUNG
   RUNG wire#powerrail
      R_Coil( "qR1ToolSelect2" )
   END_RUNG
   // the same network as SCL:
   "qR1ToolSelect1" := TRUE;
   "qR1ToolSelect2" := FALSE;
END_REGION

REGION Network 17: audio signal before safety start
   RUNG wire#powerrail
      Contact( #"ESTOP1_3L+".Q )
      I_Contact( #"F_IEC_Timer_3L+".Q )
      wire#w1
      Contact( "safety_signals".Clock_1Hz )
      Coil( "qAudioSignal" )
   END_RUNG
   RUNG wire#powerrail
      Contact( #"ESTOP1_4L+".Q )
      Contact( #"ESTOP1_3L+".Q )
      I_Contact( #"F_IEC_Timer_4L+".Q )
   END_RUNG wire#w1
   // the same network as SCL:
   "qAudioSignal" := ((#"ESTOP1_3L+".Q AND NOT #"F_IEC_Timer_3L+".Q) OR (#"ESTOP1_4L+".Q AND #"ESTOP1_3L+".Q AND NOT #"F_IEC_Timer_4L+".Q)) AND "safety_signals".Clock_1Hz;
END_REGION

REGION Network 18: hydraulic motor - EDM
   RUNG wire#powerrail
      #FDBACK_KM20_KM21.FDBACK(ON := "DevicesData".Hydraulic.StartMotor, FEEDBACK := "iEDM_KM20_KM21", QBAD_FIO :=, ACK_NEC :=, ACK := "Alarms".Reset, FDB_TIME := t#300ms, Q =>, ERROR =>, ACK_REQ =>, DIAG =>)
   END_RUNG
   // the same network as SCL:
   #FDBACK_KM20_KM21(ON := "DevicesData".Hydraulic.StartMotor,   // FDBACK
                     FEEDBACK := "iEDM_KM20_KM21",
                     ACK := "Alarms".Reset,
                     FDB_TIME := t#300ms);
END_REGION

REGION Network 19: hydraulic motor - set output
   RUNG wire#powerrail
      Contact( #FDBACK_KM20_KM21.Q )
      Coil( "qHydraulicKM20" )
      Coil( "qHydraulicKM21" )
   END_RUNG
   // the same network as SCL:
   "qHydraulicKM20" := #FDBACK_KM20_KM21.Q;
   "qHydraulicKM21" := #FDBACK_KM20_KM21.Q;
END_REGION
END_FUNCTION_BLOCK

FUNCTION_BLOCK "sq_autoeject"   // FB53, GRAPH
VERSION : 0.1
// stored: AcknowledgeErrorsRequired true, AutoNumber true, GraphVersion 6.0, InitialValuesAcquisition false, IsIECCheckEnabled false, LanguageInNetworks LAD, LockOperatingMode false, PermanentILProcessingInMANMode false, SetENOAutomatically false, SkipSteps false, UDAEnableTagReadback false, WithAlarmHandling true
   // inherited from GRAPH_BASE
   VAR
      OFF_SQ_BASE : Bool;
   END_VAR
   VAR_INPUT
      OFF_SQ { ExternalWritable := 'False'} : Bool := false;   // Turn sequence off
      INIT_SQ { ExternalWritable := 'False'} : Bool := false;   // Set sequence to initial state
      ACK_EF { ExternalWritable := 'False'} : Bool := false;   // Acknowledge all errors and faults
      S_PREV { ExternalWritable := 'False'} : Bool := false;   // Output previous step in parameter S_NO
      S_NEXT { ExternalWritable := 'False'} : Bool := false;   // Indicate next step in parameter S_NO
      SW_AUTO { ExternalWritable := 'False'} : Bool := false;   // Automatic mode
      SW_TAP { ExternalWritable := 'False'} : Bool := false;   // Semiautomatic/switch with transition
      SW_TOP { ExternalWritable := 'False'} : Bool := false;   // Semiautomatic/ignore transition
      SW_MAN { ExternalWritable := 'False'} : Bool := false;   // Manual mode
      S_SEL { ExternalWritable := 'False'} : Int := 0;   // Select step to be output to S_NO
      S_ON { ExternalWritable := 'False'} : Bool := false;   // Activate step indicated in S_NO
      S_OFF { ExternalWritable := 'False'} : Bool := false;   // Deactivate step indicated S_NO
      T_PUSH { ExternalWritable := 'False'} : Bool := false;   // Enable transition to switch in semi automatic mode
   END_VAR
   VAR_OUTPUT
      S_NO { ExternalWritable := 'False'} : Int := 0;   // Step number
      S_MORE { ExternalWritable := 'False'} : Bool := false;   // More steps are available and can be shown in S_NO
      S_ACTIVE { ExternalWritable := 'False'} : Bool := false;   // Step indicated in S_NO is active
      ERR_FLT { ExternalWritable := 'False'} : Bool := false;   // Interlock or supervision group error
      AUTO_ON { ExternalWritable := 'False'} : Bool := false;   // Automatic mode is active
      TAP_ON { ExternalWritable := 'False'} : Bool := false;   // Semiautomatic mode/step with transition enabled
      TOP_ON { ExternalWritable := 'False'} : Bool := false;   // Semiautomatic mode/ignore transition enabled
      MAN_ON { ExternalWritable := 'False'} : Bool := false;   // Manual mode is active
   END_VAR
   VAR
      dummy : Bool;
      start : Bool;
      base : Bool;
   END_VAR
BEGIN
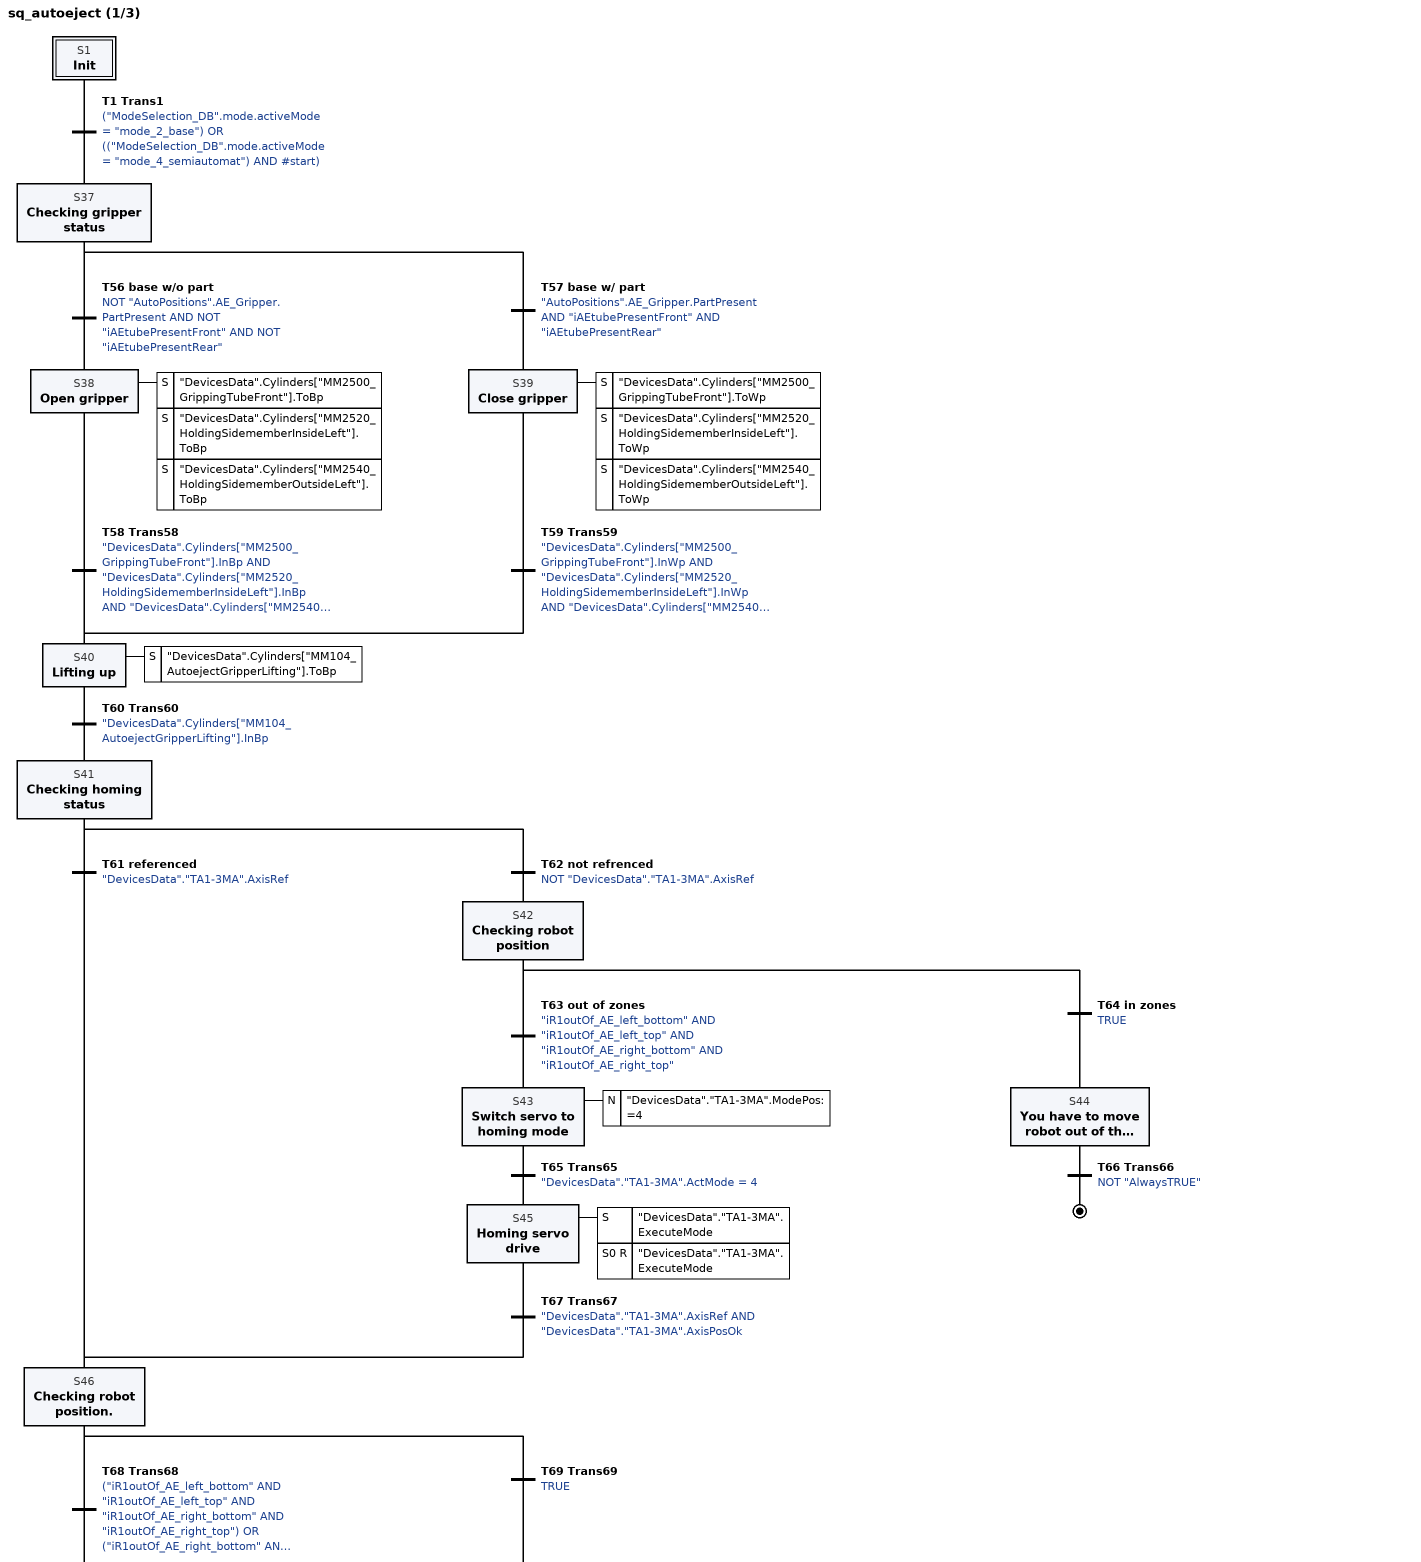
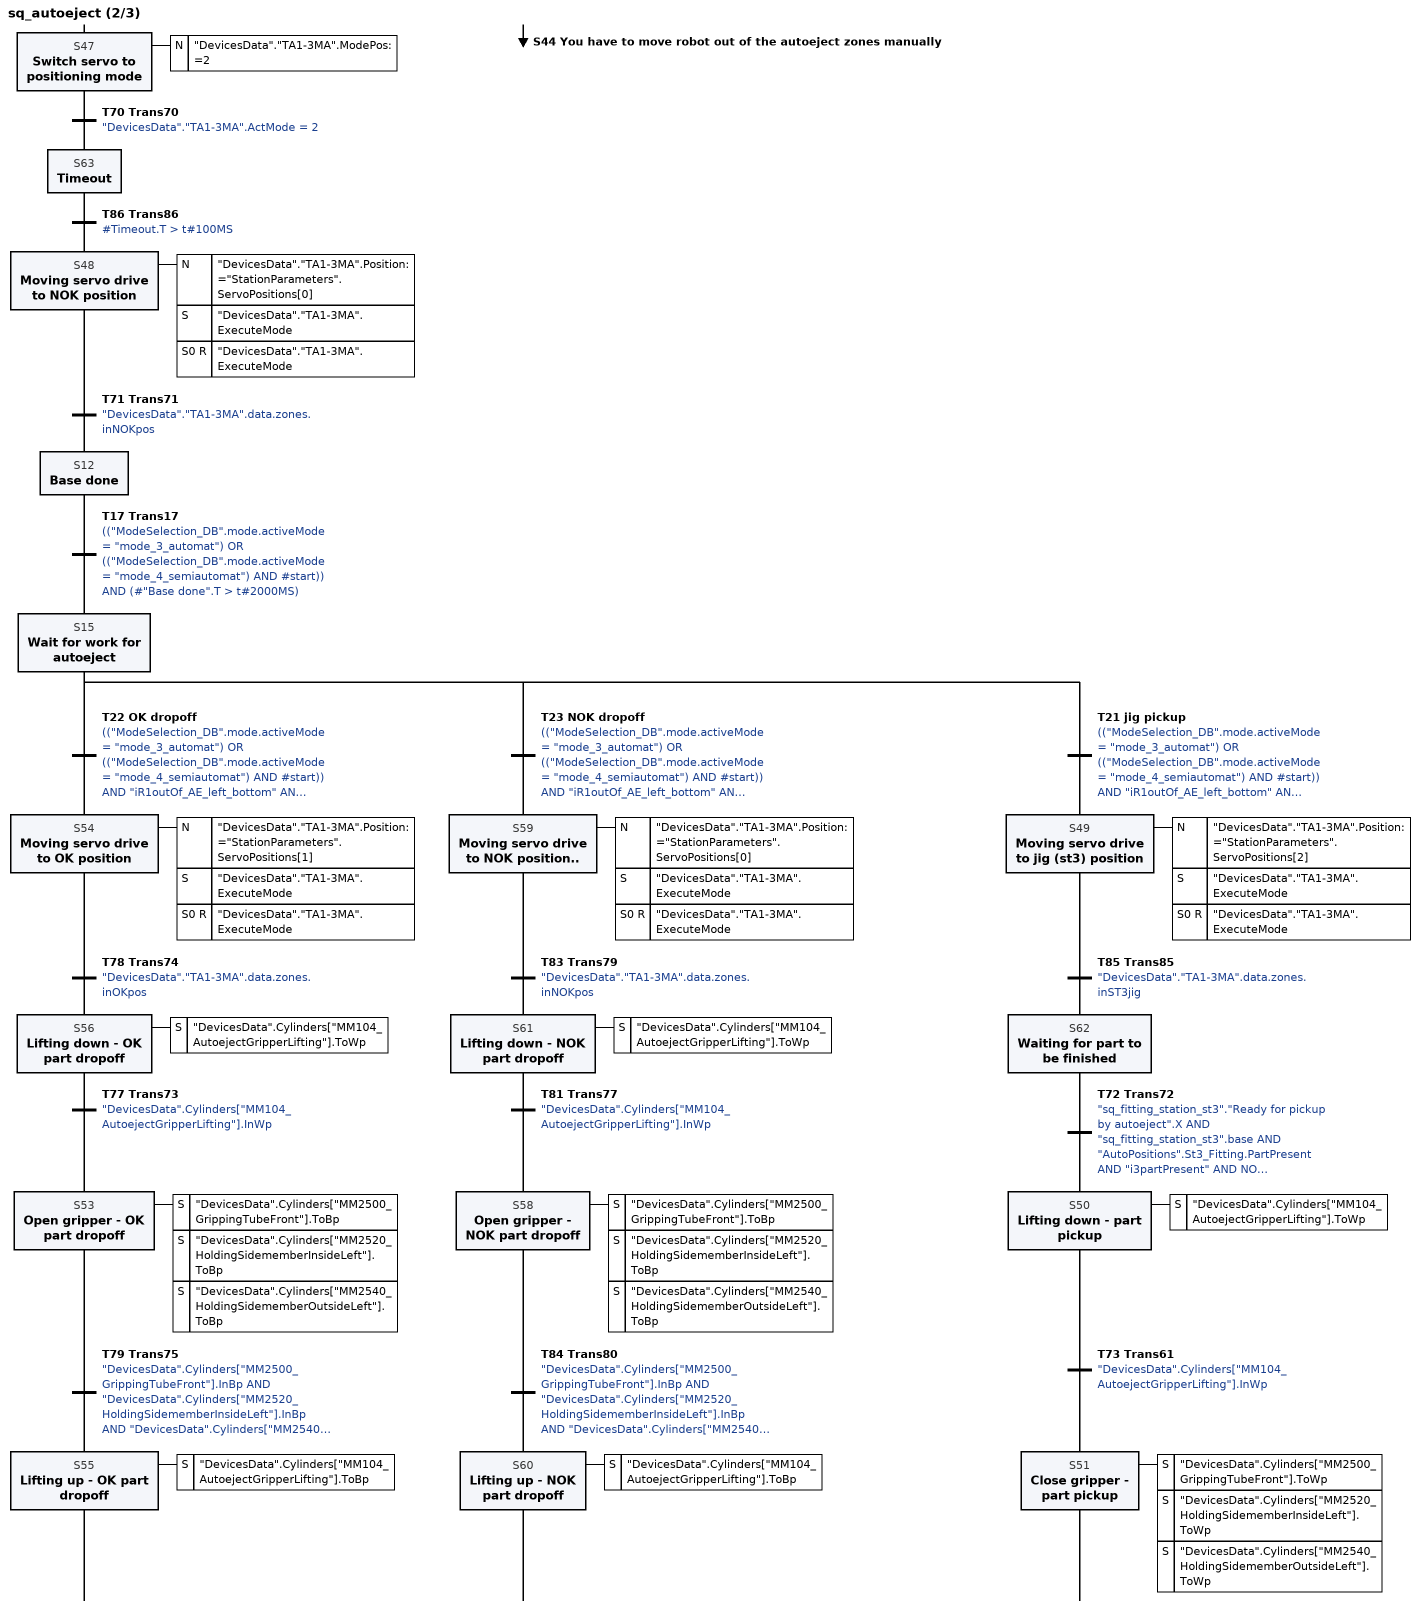
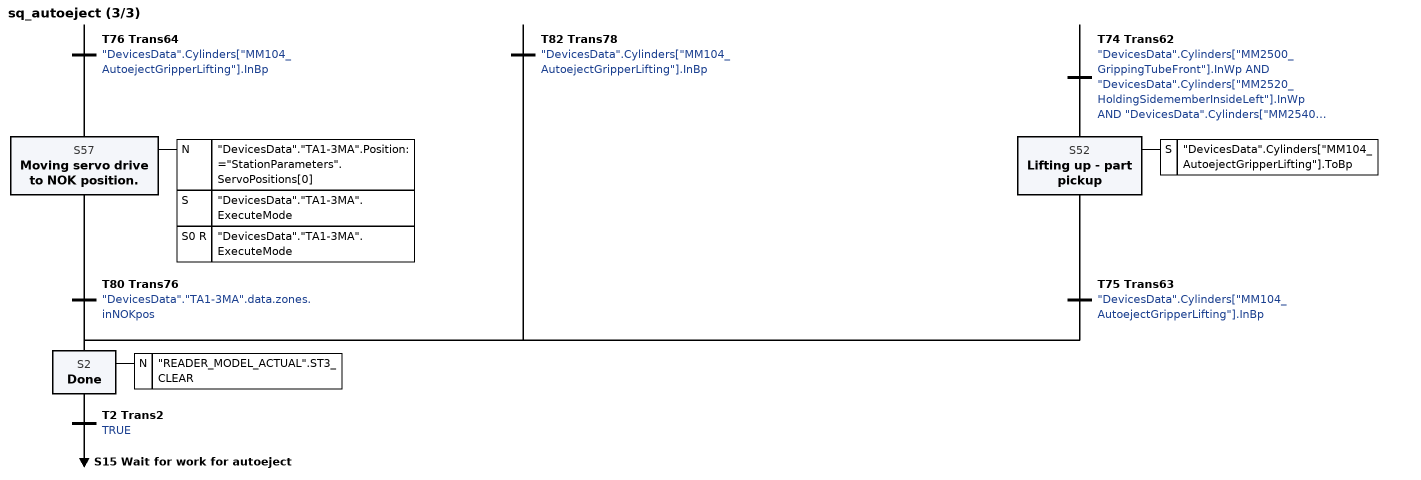
   // sequencer 1
   INITIAL_STEP Init:   // S1, max time T#10S, warning time T#7S
   END_STEP
   TRANSITION Trans1 FROM Init TO "Checking gripper status"   // T1
      := ("ModeSelection_DB".mode.activeMode = "mode_2_base") OR (("ModeSelection_DB".mode.activeMode = "mode_4_semiautomat") AND #start);
   END_TRANSITION
   STEP Done:   // S2, max time T#10S, warning time T#7S
              N    "READER_MODEL_ACTUAL".ST3_CLEAR
   END_STEP
   TRANSITION Trans2 FROM Done TO "Wait for work for autoeject"   // T2, jump
      := TRUE;
   END_TRANSITION
   STEP "Base done":   // S12, max time T#10S, warning time T#7S
   END_STEP
   TRANSITION Trans17 FROM "Base done" TO "Wait for work for autoeject"   // T17
      := (("ModeSelection_DB".mode.activeMode = "mode_3_automat") OR (("ModeSelection_DB".mode.activeMode = "mode_4_semiautomat") AND #start)) AND (#"Base done".T > t#2000MS);
   END_TRANSITION
   STEP "Wait for work for autoeject":   // S15, max time T#10S, warning time T#7S
   END_STEP
   TRANSITION "OK dropoff" FROM "Wait for work for autoeject" TO "Moving servo drive to OK position"   // T22
      := (("ModeSelection_DB".mode.activeMode = "mode_3_automat") OR (("ModeSelection_DB".mode.activeMode = "mode_4_semiautomat") AND #start)) AND "iR1outOf_AE_left_bottom" AND "iR1outOf_AE_left_top" AND "iR1outOf_AE_right_bottom" AND "iR1outOf_AE_right_top" AND "AutoPositions".AE_Gripper.PartPresent AND "AutoPositions".AE_Gripper.StFinished[3] AND NOT "AutoPositions".AE_Gripper.PartNOK AND "iAEtubePresentFront" AND "iAEtubePresentRear" AND NOT "AutoPositions".St4_OKposition.PartPresent AND NOT "i4partPresent";
   END_TRANSITION
   TRANSITION "NOK dropoff" FROM "Wait for work for autoeject" TO "Moving servo drive to NOK position.."   // T23
      := (("ModeSelection_DB".mode.activeMode = "mode_3_automat") OR (("ModeSelection_DB".mode.activeMode = "mode_4_semiautomat") AND #start)) AND "iR1outOf_AE_left_bottom" AND "iR1outOf_AE_left_top" AND "iR1outOf_AE_right_bottom" AND "iR1outOf_AE_right_top" AND "AutoPositions".AE_Gripper.PartPresent AND (NOT "AutoPositions".AE_Gripper.StFinished[3] OR "AutoPositions".AE_Gripper.PartNOK) AND "iAEtubePresentFront" AND "iAEtubePresentRear" AND NOT "PartHolderData".NOKBoxFull;
   END_TRANSITION
   TRANSITION "jig pickup" FROM "Wait for work for autoeject" TO "Moving servo drive to jig (st3) position"   // T21
      := (("ModeSelection_DB".mode.activeMode = "mode_3_automat") OR (("ModeSelection_DB".mode.activeMode = "mode_4_semiautomat") AND #start)) AND "iR1outOf_AE_left_bottom" AND "iR1outOf_AE_left_top" AND "iR1outOf_AE_right_bottom" AND "iR1outOf_AE_right_top" AND "AutoPositions".St3_Fitting.PartPresent AND "i3partPresent" AND NOT "AutoPositions".AE_Gripper.PartPresent AND NOT "iAEtubePresentFront" AND NOT "iAEtubePresentRear" AND NOT "AutoPositions".St4_OKposition.PartPresent AND NOT "i4partPresent";
   END_TRANSITION
   STEP "Close gripper - part pickup":   // S51, max time T#10S, warning time T#7S
              S    "DevicesData".Cylinders["MM2500_GrippingTubeFront"].ToWp
              S    "DevicesData".Cylinders["MM2520_HoldingSidememberInsideLeft"].ToWp
              S    "DevicesData".Cylinders["MM2540_HoldingSidememberOutsideLeft"].ToWp
   END_STEP
   TRANSITION Trans62 FROM "Close gripper - part pickup" TO "Lifting up - part pickup"   // T74
      := "DevicesData".Cylinders["MM2500_GrippingTubeFront"].InWp AND "DevicesData".Cylinders["MM2520_HoldingSidememberInsideLeft"].InWp AND "DevicesData".Cylinders["MM2540_HoldingSidememberOutsideLeft"].InWp;
   END_TRANSITION
   STEP "Open gripper - OK part dropoff":   // S53, max time T#10S, warning time T#7S
              S    "DevicesData".Cylinders["MM2500_GrippingTubeFront"].ToBp
              S    "DevicesData".Cylinders["MM2520_HoldingSidememberInsideLeft"].ToBp
              S    "DevicesData".Cylinders["MM2540_HoldingSidememberOutsideLeft"].ToBp
   END_STEP
   TRANSITION Trans75 FROM "Open gripper - OK part dropoff" TO "Lifting up - OK part dropoff"   // T79
      := "DevicesData".Cylinders["MM2500_GrippingTubeFront"].InBp AND "DevicesData".Cylinders["MM2520_HoldingSidememberInsideLeft"].InBp AND "DevicesData".Cylinders["MM2540_HoldingSidememberOutsideLeft"].InBp;
   END_TRANSITION
   STEP "Moving servo drive to OK position":   // S54, max time T#30S, warning time T#7S
      supervision V := #"Moving servo drive to OK position".T > #"Moving servo drive to OK position".T_MAX;
              N    "DevicesData"."TA1-3MA".Position:="StationParameters".ServoPositions[1]
              S    "DevicesData"."TA1-3MA".ExecuteMode
          S0  R    "DevicesData"."TA1-3MA".ExecuteMode
   END_STEP
   TRANSITION Trans74 FROM "Moving servo drive to OK position" TO "Lifting down - OK part dropoff"   // T78
      := "DevicesData"."TA1-3MA".data.zones.inOKpos;
   END_TRANSITION
   STEP "Lifting up - OK part dropoff":   // S55, max time T#10S, warning time T#7S
              S    "DevicesData".Cylinders["MM104_AutoejectGripperLifting"].ToBp
   END_STEP
   TRANSITION Trans64 FROM "Lifting up - OK part dropoff" TO "Moving servo drive to NOK position."   // T76
      := "DevicesData".Cylinders["MM104_AutoejectGripperLifting"].InBp;
   END_TRANSITION
   STEP "Lifting down - OK part dropoff":   // S56, max time T#10S, warning time T#7S
              S    "DevicesData".Cylinders["MM104_AutoejectGripperLifting"].ToWp
   END_STEP
   TRANSITION Trans73 FROM "Lifting down - OK part dropoff" TO "Open gripper - OK part dropoff"   // T77
      := "DevicesData".Cylinders["MM104_AutoejectGripperLifting"].InWp;
   END_TRANSITION
   STEP "Moving servo drive to jig (st3) position":   // S49, max time T#30S, warning time T#7S
      supervision V := #"Moving servo drive to jig (st3) position".T > #"Moving servo drive to jig (st3) position".T_MAX;
              N    "DevicesData"."TA1-3MA".Position:="StationParameters".ServoPositions[2]
              S    "DevicesData"."TA1-3MA".ExecuteMode
          S0  R    "DevicesData"."TA1-3MA".ExecuteMode
   END_STEP
   TRANSITION Trans85 FROM "Moving servo drive to jig (st3) position" TO "Waiting for part to be finished"   // T85
      := "DevicesData"."TA1-3MA".data.zones.inST3jig;
   END_TRANSITION
   STEP "Lifting up - part pickup":   // S52, max time T#10S, warning time T#7S
              S    "DevicesData".Cylinders["MM104_AutoejectGripperLifting"].ToBp
   END_STEP
   TRANSITION Trans63 FROM "Lifting up - part pickup" TO Done   // T75
      := "DevicesData".Cylinders["MM104_AutoejectGripperLifting"].InBp;
   END_TRANSITION
   STEP "Lifting down - part pickup":   // S50, max time T#10S, warning time T#7S
              S    "DevicesData".Cylinders["MM104_AutoejectGripperLifting"].ToWp
   END_STEP
   TRANSITION Trans61 FROM "Lifting down - part pickup" TO "Close gripper - part pickup"   // T73
      := "DevicesData".Cylinders["MM104_AutoejectGripperLifting"].InWp;
   END_TRANSITION
   STEP "Checking gripper status":   // S37, max time T#10S, warning time T#7S
   END_STEP
   TRANSITION "base w/o part" FROM "Checking gripper status" TO "Open gripper"   // T56
      := NOT "AutoPositions".AE_Gripper.PartPresent AND NOT "iAEtubePresentFront" AND NOT "iAEtubePresentRear";
   END_TRANSITION
   TRANSITION "base w/ part" FROM "Checking gripper status" TO "Close gripper"   // T57
      := "AutoPositions".AE_Gripper.PartPresent AND "iAEtubePresentFront" AND "iAEtubePresentRear";
   END_TRANSITION
   STEP "Open gripper":   // S38, max time T#10S, warning time T#7S
              S    "DevicesData".Cylinders["MM2500_GrippingTubeFront"].ToBp
              S    "DevicesData".Cylinders["MM2520_HoldingSidememberInsideLeft"].ToBp
              S    "DevicesData".Cylinders["MM2540_HoldingSidememberOutsideLeft"].ToBp
   END_STEP
   TRANSITION Trans58 FROM "Open gripper" TO "Lifting up"   // T58
      := "DevicesData".Cylinders["MM2500_GrippingTubeFront"].InBp AND "DevicesData".Cylinders["MM2520_HoldingSidememberInsideLeft"].InBp AND "DevicesData".Cylinders["MM2540_HoldingSidememberOutsideLeft"].InBp;
   END_TRANSITION
   STEP "Close gripper":   // S39, max time T#10S, warning time T#7S
              S    "DevicesData".Cylinders["MM2500_GrippingTubeFront"].ToWp
              S    "DevicesData".Cylinders["MM2520_HoldingSidememberInsideLeft"].ToWp
              S    "DevicesData".Cylinders["MM2540_HoldingSidememberOutsideLeft"].ToWp
   END_STEP
   TRANSITION Trans59 FROM "Close gripper" TO "Lifting up"   // T59
      := "DevicesData".Cylinders["MM2500_GrippingTubeFront"].InWp AND "DevicesData".Cylinders["MM2520_HoldingSidememberInsideLeft"].InWp AND "DevicesData".Cylinders["MM2540_HoldingSidememberOutsideLeft"].InWp;
   END_TRANSITION
   STEP "Lifting up":   // S40, max time T#10S, warning time T#7S
              S    "DevicesData".Cylinders["MM104_AutoejectGripperLifting"].ToBp
   END_STEP
   TRANSITION Trans60 FROM "Lifting up" TO "Checking homing status"   // T60
      := "DevicesData".Cylinders["MM104_AutoejectGripperLifting"].InBp;
   END_TRANSITION
   STEP "Checking homing status":   // S41, max time T#10S, warning time T#7S
   END_STEP
   TRANSITION referenced FROM "Checking homing status" TO "Checking robot position."   // T61
      := "DevicesData"."TA1-3MA".AxisRef;
   END_TRANSITION
   TRANSITION "not refrenced" FROM "Checking homing status" TO "Checking robot position"   // T62
      := NOT "DevicesData"."TA1-3MA".AxisRef;
   END_TRANSITION
   STEP "Checking robot position":   // S42, max time T#10S, warning time T#7S
   END_STEP
   TRANSITION "out of zones" FROM "Checking robot position" TO "Switch servo to homing mode"   // T63
      := "iR1outOf_AE_left_bottom" AND "iR1outOf_AE_left_top" AND "iR1outOf_AE_right_bottom" AND "iR1outOf_AE_right_top";
   END_TRANSITION
   TRANSITION "in zones" FROM "Checking robot position" TO "You have to move robot out of the autoeject zones manually"   // T64
      := TRUE;
   END_TRANSITION
   STEP "Switch servo to homing mode":   // S43, max time T#10S, warning time T#7S
      supervision V := #"Switch servo to homing mode".T > #"Switch servo to homing mode".T_MAX;
              N    "DevicesData"."TA1-3MA".ModePos:=4
   END_STEP
   TRANSITION Trans65 FROM "Switch servo to homing mode" TO "Homing servo drive"   // T65
      := "DevicesData"."TA1-3MA".ActMode = 4;
   END_TRANSITION
   STEP "You have to move robot out of the autoeject zones manually":   // S44, max time T#10S, warning time T#7S
      supervision V := "AlwaysTRUE";
   END_STEP
   TRANSITION Trans66 FROM "You have to move robot out of the autoeject zones manually" TO END   // T66
      := NOT "AlwaysTRUE";
   END_TRANSITION
   STEP "Homing servo drive":   // S45, max time T#30S, warning time T#7S
      supervision V := #"Homing servo drive".T > #"Homing servo drive".T_MAX;
              S    "DevicesData"."TA1-3MA".ExecuteMode
          S0  R    "DevicesData"."TA1-3MA".ExecuteMode
   END_STEP
   TRANSITION Trans67 FROM "Homing servo drive" TO "Checking robot position."   // T67
      := "DevicesData"."TA1-3MA".AxisRef AND "DevicesData"."TA1-3MA".AxisPosOk;
   END_TRANSITION
   STEP "Checking robot position.":   // S46, max time T#10S, warning time T#7S
   END_STEP
   TRANSITION Trans68 FROM "Checking robot position." TO "Switch servo to positioning mode"   // T68
      := ("iR1outOf_AE_left_bottom" AND "iR1outOf_AE_left_top" AND "iR1outOf_AE_right_bottom" AND "iR1outOf_AE_right_top") OR ("iR1outOf_AE_right_bottom" AND "iR1outOf_AE_right_top" AND "DevicesData"."TA1-3MA".data.zones.outOfST3zone);
   END_TRANSITION
   TRANSITION Trans69 FROM "Checking robot position." TO "You have to move robot out of the autoeject zones manually"   // T69, jump
      := TRUE;
   END_TRANSITION
   STEP "Switch servo to positioning mode":   // S47, max time T#10S, warning time T#7S
      supervision V := #"Switch servo to positioning mode".T > #"Switch servo to positioning mode".T_MAX;
              N    "DevicesData"."TA1-3MA".ModePos:=2
   END_STEP
   TRANSITION Trans70 FROM "Switch servo to positioning mode" TO Timeout   // T70
      := "DevicesData"."TA1-3MA".ActMode = 2;
   END_TRANSITION
   STEP "Moving servo drive to NOK position":   // S48, max time T#30S, warning time T#7S
      supervision V := #"Moving servo drive to NOK position".T > #"Moving servo drive to NOK position".T_MAX;
              N    "DevicesData"."TA1-3MA".Position:="StationParameters".ServoPositions[0]
              S    "DevicesData"."TA1-3MA".ExecuteMode
          S0  R    "DevicesData"."TA1-3MA".ExecuteMode
   END_STEP
   TRANSITION Trans71 FROM "Moving servo drive to NOK position" TO "Base done"   // T71
      := "DevicesData"."TA1-3MA".data.zones.inNOKpos;
   END_TRANSITION
   STEP "Moving servo drive to NOK position.":   // S57, max time T#30S, warning time T#7S
      supervision V := #"Moving servo drive to NOK position.".T > #"Moving servo drive to NOK position.".T_MAX;
              N    "DevicesData"."TA1-3MA".Position:="StationParameters".ServoPositions[0]
              S    "DevicesData"."TA1-3MA".ExecuteMode
          S0  R    "DevicesData"."TA1-3MA".ExecuteMode
   END_STEP
   TRANSITION Trans76 FROM "Moving servo drive to NOK position." TO Done   // T80
      := "DevicesData"."TA1-3MA".data.zones.inNOKpos;
   END_TRANSITION
   STEP "Open gripper - NOK part dropoff":   // S58, max time T#10S, warning time T#7S
              S    "DevicesData".Cylinders["MM2500_GrippingTubeFront"].ToBp
              S    "DevicesData".Cylinders["MM2520_HoldingSidememberInsideLeft"].ToBp
              S    "DevicesData".Cylinders["MM2540_HoldingSidememberOutsideLeft"].ToBp
   END_STEP
   TRANSITION Trans80 FROM "Open gripper - NOK part dropoff" TO "Lifting up - NOK part dropoff"   // T84
      := "DevicesData".Cylinders["MM2500_GrippingTubeFront"].InBp AND "DevicesData".Cylinders["MM2520_HoldingSidememberInsideLeft"].InBp AND "DevicesData".Cylinders["MM2540_HoldingSidememberOutsideLeft"].InBp;
   END_TRANSITION
   STEP "Moving servo drive to NOK position..":   // S59, max time T#30S, warning time T#7S
      supervision V := #"Moving servo drive to NOK position..".T > #"Moving servo drive to NOK position..".T_MAX;
              N    "DevicesData"."TA1-3MA".Position:="StationParameters".ServoPositions[0]
              S    "DevicesData"."TA1-3MA".ExecuteMode
          S0  R    "DevicesData"."TA1-3MA".ExecuteMode
   END_STEP
   TRANSITION Trans79 FROM "Moving servo drive to NOK position.." TO "Lifting down - NOK part dropoff"   // T83
      := "DevicesData"."TA1-3MA".data.zones.inNOKpos;
   END_TRANSITION
   STEP "Lifting up - NOK part dropoff":   // S60, max time T#10S, warning time T#7S
              S    "DevicesData".Cylinders["MM104_AutoejectGripperLifting"].ToBp
   END_STEP
   TRANSITION Trans78 FROM "Lifting up - NOK part dropoff" TO Done   // T82
      := "DevicesData".Cylinders["MM104_AutoejectGripperLifting"].InBp;
   END_TRANSITION
   STEP "Lifting down - NOK part dropoff":   // S61, max time T#10S, warning time T#7S
              S    "DevicesData".Cylinders["MM104_AutoejectGripperLifting"].ToWp
   END_STEP
   TRANSITION Trans77 FROM "Lifting down - NOK part dropoff" TO "Open gripper - NOK part dropoff"   // T81
      := "DevicesData".Cylinders["MM104_AutoejectGripperLifting"].InWp;
   END_TRANSITION
   STEP "Waiting for part to be finished":   // S62, max time T#10S, warning time T#7S
   END_STEP
   TRANSITION Trans72 FROM "Waiting for part to be finished" TO "Lifting down - part pickup"   // T72
      := "sq_fitting_station_st3"."Ready for pickup by autoeject".X AND "sq_fitting_station_st3".base AND "AutoPositions".St3_Fitting.PartPresent AND "i3partPresent" AND NOT "AutoPositions".AE_Gripper.PartPresent AND NOT "iAEtubePresentFront" AND NOT "iAEtubePresentRear" AND NOT "AutoPositions".St4_OKposition.PartPresent;
   END_TRANSITION
   STEP Timeout:   // S63, max time T#10S, warning time T#7S
   END_STEP
   TRANSITION Trans86 FROM Timeout TO "Moving servo drive to NOK position"   // T86
      := #Timeout.T > t#100MS;
   END_TRANSITION
END_FUNCTION_BLOCK

FUNCTION_BLOCK "sq_carousel_main"   // FB70, GRAPH
VERSION : 0.1
// stored: AcknowledgeErrorsRequired true, AutoNumber true, GraphVersion 6.0, InitialValuesAcquisition false, IsIECCheckEnabled false, LanguageInNetworks LAD, LockOperatingMode false, PermanentILProcessingInMANMode false, SetENOAutomatically false, SkipSteps false, UDAEnableTagReadback false, WithAlarmHandling true
   // inherited from GRAPH_BASE
   VAR
      OFF_SQ_BASE : Bool;
   END_VAR
   VAR_INPUT
      OFF_SQ { ExternalAccessible := 'False'; ExternalVisible := 'False'; ExternalWritable := 'False'} : Bool := false;   // Turn sequence off
      INIT_SQ { ExternalAccessible := 'False'; ExternalVisible := 'False'; ExternalWritable := 'False'} : Bool := false;   // Set sequence to initial state
      ACK_EF { ExternalAccessible := 'False'; ExternalVisible := 'False'; ExternalWritable := 'False'} : Bool := false;   // Acknowledge all errors and faults
      S_PREV { ExternalAccessible := 'False'; ExternalVisible := 'False'; ExternalWritable := 'False'} : Bool := false;   // Output previous step in parameter S_NO
      S_NEXT { ExternalAccessible := 'False'; ExternalVisible := 'False'; ExternalWritable := 'False'} : Bool := false;   // Indicate next step in parameter S_NO
      SW_AUTO { ExternalAccessible := 'False'; ExternalVisible := 'False'; ExternalWritable := 'False'} : Bool := false;   // Automatic mode
      SW_TAP { ExternalAccessible := 'False'; ExternalVisible := 'False'; ExternalWritable := 'False'} : Bool := false;   // Semiautomatic/switch with transition
      SW_TOP { ExternalAccessible := 'False'; ExternalVisible := 'False'; ExternalWritable := 'False'} : Bool := false;   // Semiautomatic/ignore transition
      SW_MAN { ExternalAccessible := 'False'; ExternalVisible := 'False'; ExternalWritable := 'False'} : Bool := false;   // Manual mode
      S_SEL { ExternalAccessible := 'False'; ExternalVisible := 'False'; ExternalWritable := 'False'} : Int := 0;   // Select step to be output to S_NO
      S_ON { ExternalAccessible := 'False'; ExternalVisible := 'False'; ExternalWritable := 'False'} : Bool := false;   // Activate step indicated in S_NO
      S_OFF { ExternalAccessible := 'False'; ExternalVisible := 'False'; ExternalWritable := 'False'} : Bool := false;   // Deactivate step indicated S_NO
      T_PUSH { ExternalAccessible := 'False'; ExternalVisible := 'False'; ExternalWritable := 'False'} : Bool := false;   // Enable transition to switch in semi automatic mode
   END_VAR
   VAR_OUTPUT
      S_NO { ExternalAccessible := 'False'; ExternalVisible := 'False'; ExternalWritable := 'False'} : Int := 0;   // Step number
      S_MORE { ExternalAccessible := 'False'; ExternalVisible := 'False'; ExternalWritable := 'False'} : Bool := false;   // More steps are available and can be shown in S_NO
      S_ACTIVE { ExternalAccessible := 'False'; ExternalVisible := 'False'; ExternalWritable := 'False'} : Bool := false;   // Step indicated in S_NO is active
      ERR_FLT { ExternalAccessible := 'False'; ExternalVisible := 'False'; ExternalWritable := 'False'} : Bool := false;   // Interlock or supervision group error
      AUTO_ON { ExternalAccessible := 'False'; ExternalVisible := 'False'; ExternalWritable := 'False'} : Bool := false;   // Automatic mode is active
      TAP_ON { ExternalAccessible := 'False'; ExternalVisible := 'False'; ExternalWritable := 'False'} : Bool := false;   // Semiautomatic mode/step with transition enabled
      TOP_ON { ExternalAccessible := 'False'; ExternalVisible := 'False'; ExternalWritable := 'False'} : Bool := false;   // Semiautomatic mode/ignore transition enabled
      MAN_ON { ExternalAccessible := 'False'; ExternalVisible := 'False'; ExternalWritable := 'False'} : Bool := false;   // Manual mode is active
   END_VAR
   VAR
      dummy : Bool;
      start : Bool;
      base : Bool;
   END_VAR
BEGIN
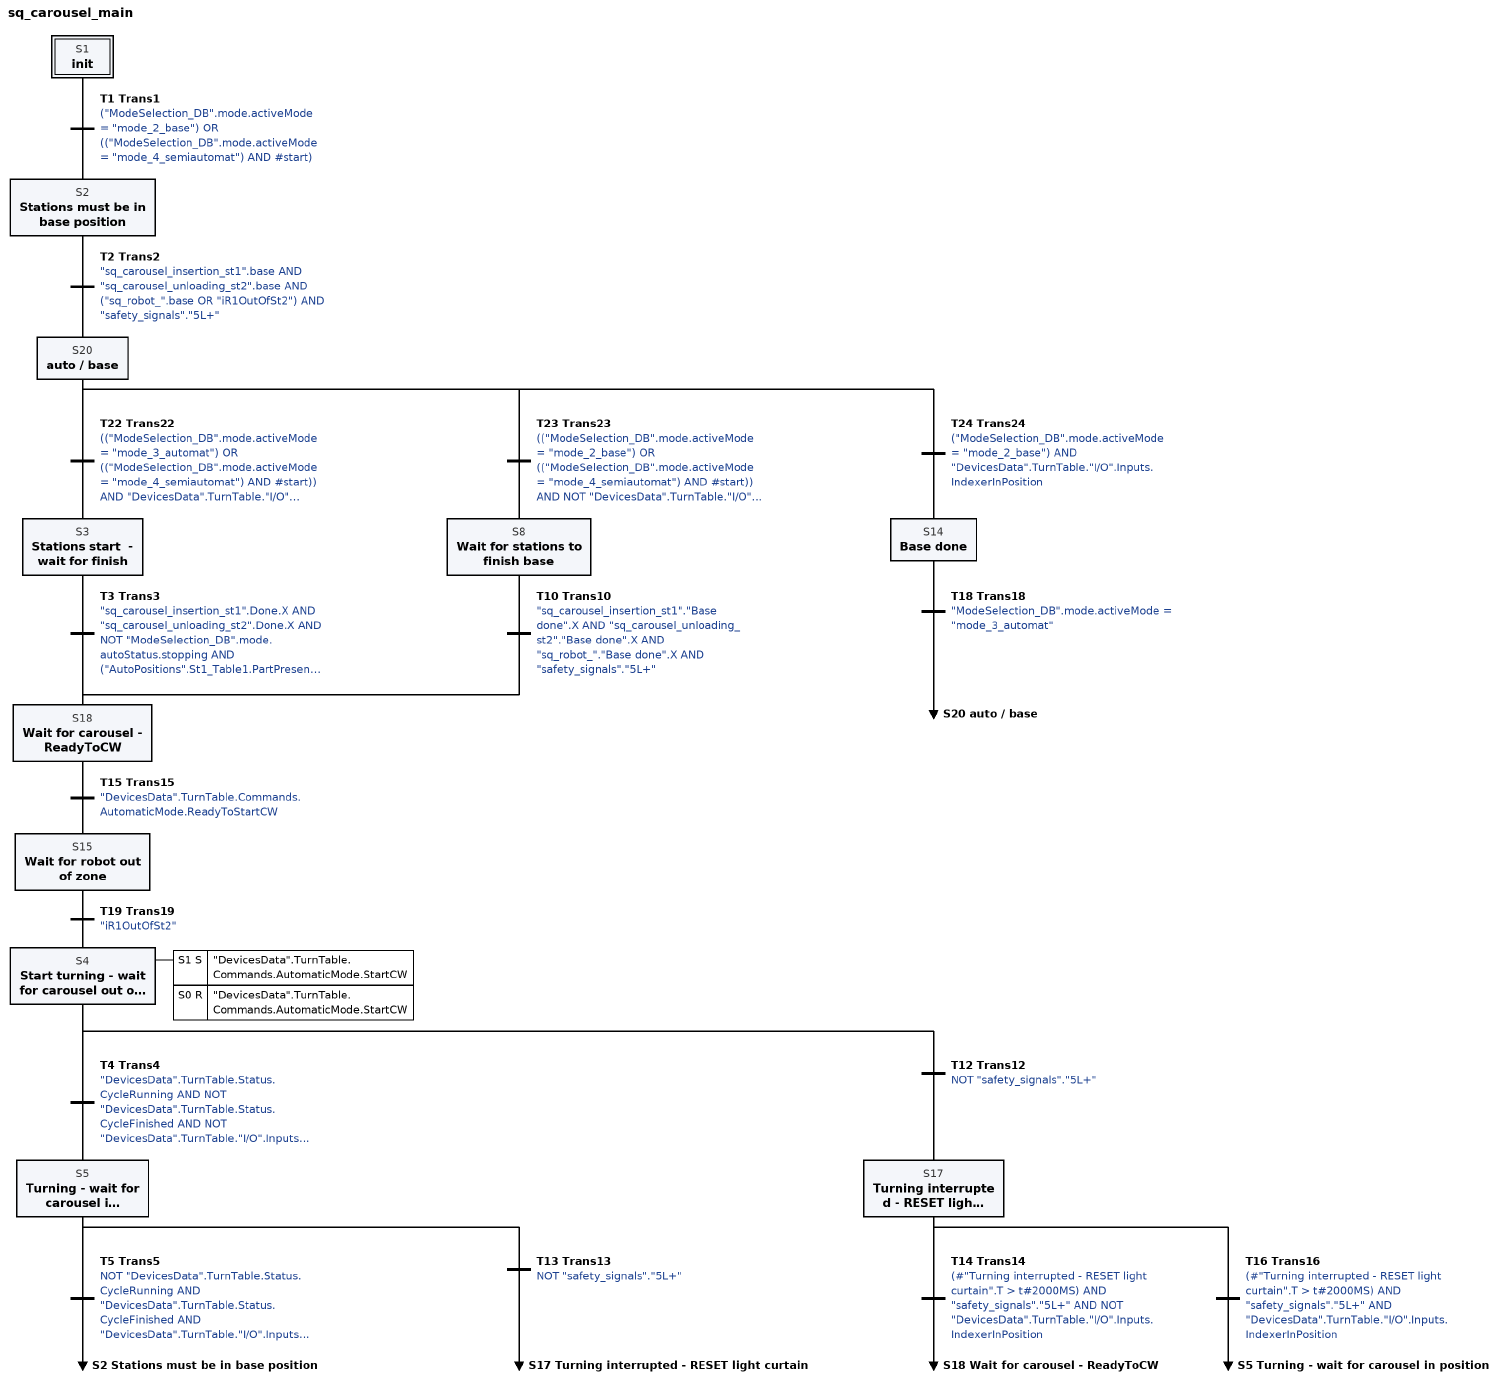
   // permanent pre-instructions
   NETWORK 1
      #base := "iTurnTableIndexerInPosition";

   // sequencer 1
   INITIAL_STEP init:   // S1, max time T#10S, warning time T#7S
   END_STEP
   TRANSITION Trans1 FROM init TO "Stations must be in base position"   // T1
      := ("ModeSelection_DB".mode.activeMode = "mode_2_base") OR (("ModeSelection_DB".mode.activeMode = "mode_4_semiautomat") AND #start);
   END_TRANSITION
   STEP "Stations must be in base position":   // S2, max time T#10S, warning time T#7S
      supervision V := #"Stations must be in base position".T > #"Stations must be in base position".T_MAX;
   END_STEP
   TRANSITION Trans2 FROM "Stations must be in base position" TO "auto / base"   // T2
      := "sq_carousel_insertion_st1".base AND "sq_carousel_unloading_st2".base AND ("sq_robot_".base OR "iR1OutOfSt2") AND "safety_signals"."5L+";
   END_TRANSITION
   STEP "Stations start  - wait for finish":   // S3, max time T#10S, warning time T#7S
   END_STEP
   TRANSITION Trans3 FROM "Stations start  - wait for finish" TO "Wait for carousel - ReadyToCW"   // T3
      := "sq_carousel_insertion_st1".Done.X AND "sq_carousel_unloading_st2".Done.X AND NOT "ModeSelection_DB".mode.autoStatus.stopping AND ("AutoPositions".St1_Table1.PartPresent OR "AutoPositions".St2_Table2.PartPresent OR NOT "ModeSelection_DB".mode.autoStatus.emptying) AND "safety_signals"."5L+";
   END_TRANSITION
   STEP "Start turning - wait for carousel out of position":   // S4, max time T#10S, warning time T#7S
      supervision V := #"Start turning - wait for carousel out of position".T > #"Start turning - wait for carousel out of position".T_MAX;
          S1  S    "DevicesData".TurnTable.Commands.AutomaticMode.StartCW
          S0  R    "DevicesData".TurnTable.Commands.AutomaticMode.StartCW
   END_STEP
   TRANSITION Trans4 FROM "Start turning - wait for carousel out of position" TO "Turning - wait for carousel in position"   // T4
      := "DevicesData".TurnTable.Status.CycleRunning AND NOT "DevicesData".TurnTable.Status.CycleFinished AND NOT "DevicesData".TurnTable."I/O".Inputs.IndexerInPosition;
   END_TRANSITION
   TRANSITION Trans12 FROM "Start turning - wait for carousel out of position" TO "Turning interrupted - RESET light curtain"   // T12
      := NOT "safety_signals"."5L+";
   END_TRANSITION
   STEP "Turning - wait for carousel in position":   // S5, max time T#10S, warning time T#7S
      supervision V := #"Turning - wait for carousel in position".T > #"Turning - wait for carousel in position".T_MAX;
   END_STEP
   TRANSITION Trans5 FROM "Turning - wait for carousel in position" TO "Stations must be in base position"   // T5, jump
      := NOT "DevicesData".TurnTable.Status.CycleRunning AND "DevicesData".TurnTable.Status.CycleFinished AND "DevicesData".TurnTable."I/O".Inputs.IndexerInPosition;
   END_TRANSITION
   TRANSITION Trans13 FROM "Turning - wait for carousel in position" TO "Turning interrupted - RESET light curtain"   // T13, jump
      := NOT "safety_signals"."5L+";
   END_TRANSITION
   STEP "Turning interrupted - RESET light curtain":   // S17, max time T#10S, warning time T#7S
   END_STEP
   TRANSITION Trans14 FROM "Turning interrupted - RESET light curtain" TO "Wait for carousel - ReadyToCW"   // T14, jump
      := (#"Turning interrupted - RESET light curtain".T > t#2000MS) AND "safety_signals"."5L+" AND NOT "DevicesData".TurnTable."I/O".Inputs.IndexerInPosition;
   END_TRANSITION
   TRANSITION Trans16 FROM "Turning interrupted - RESET light curtain" TO "Turning - wait for carousel in position"   // T16, jump
      := (#"Turning interrupted - RESET light curtain".T > t#2000MS) AND "safety_signals"."5L+" AND "DevicesData".TurnTable."I/O".Inputs.IndexerInPosition;
   END_TRANSITION
   STEP "Wait for carousel - ReadyToCW":   // S18, max time T#10S, warning time T#7S
      supervision V := #"Wait for carousel - ReadyToCW".T > #"Wait for carousel - ReadyToCW".T_MAX;
   END_STEP
   TRANSITION Trans15 FROM "Wait for carousel - ReadyToCW" TO "Wait for robot out of zone"   // T15
      := "DevicesData".TurnTable.Commands.AutomaticMode.ReadyToStartCW;
   END_TRANSITION
   STEP "Wait for stations to finish base":   // S8, max time T#10S, warning time T#7S
   END_STEP
   TRANSITION Trans10 FROM "Wait for stations to finish base" TO "Wait for carousel - ReadyToCW"   // T10
      := "sq_carousel_insertion_st1"."Base done".X AND "sq_carousel_unloading_st2"."Base done".X AND "sq_robot_"."Base done".X AND "safety_signals"."5L+";
   END_TRANSITION
   STEP "auto / base":   // S20, max time T#10S, warning time T#7S
   END_STEP
   TRANSITION Trans22 FROM "auto / base" TO "Stations start  - wait for finish"   // T22
      := (("ModeSelection_DB".mode.activeMode = "mode_3_automat") OR (("ModeSelection_DB".mode.activeMode = "mode_4_semiautomat") AND #start)) AND "DevicesData".TurnTable."I/O".Inputs.IndexerInPosition;
   END_TRANSITION
   TRANSITION Trans23 FROM "auto / base" TO "Wait for stations to finish base"   // T23
      := (("ModeSelection_DB".mode.activeMode = "mode_2_base") OR (("ModeSelection_DB".mode.activeMode = "mode_4_semiautomat") AND #start)) AND NOT "DevicesData".TurnTable."I/O".Inputs.IndexerInPosition;
   END_TRANSITION
   TRANSITION Trans24 FROM "auto / base" TO "Base done"   // T24
      := ("ModeSelection_DB".mode.activeMode = "mode_2_base") AND "DevicesData".TurnTable."I/O".Inputs.IndexerInPosition;
   END_TRANSITION
   STEP "Base done":   // S14, max time T#10S, warning time T#7S
   END_STEP
   TRANSITION Trans18 FROM "Base done" TO "auto / base"   // T18, jump
      := "ModeSelection_DB".mode.activeMode = "mode_3_automat";
   END_TRANSITION
   STEP "Wait for robot out of zone":   // S15, max time T#10S, warning time T#7S
      supervision V := #"Wait for robot out of zone".T > #"Wait for robot out of zone".T_MAX;
   END_STEP
   TRANSITION Trans19 FROM "Wait for robot out of zone" TO "Start turning - wait for carousel out of position"   // T19
      := "iR1OutOfSt2";
   END_TRANSITION
END_FUNCTION_BLOCK

